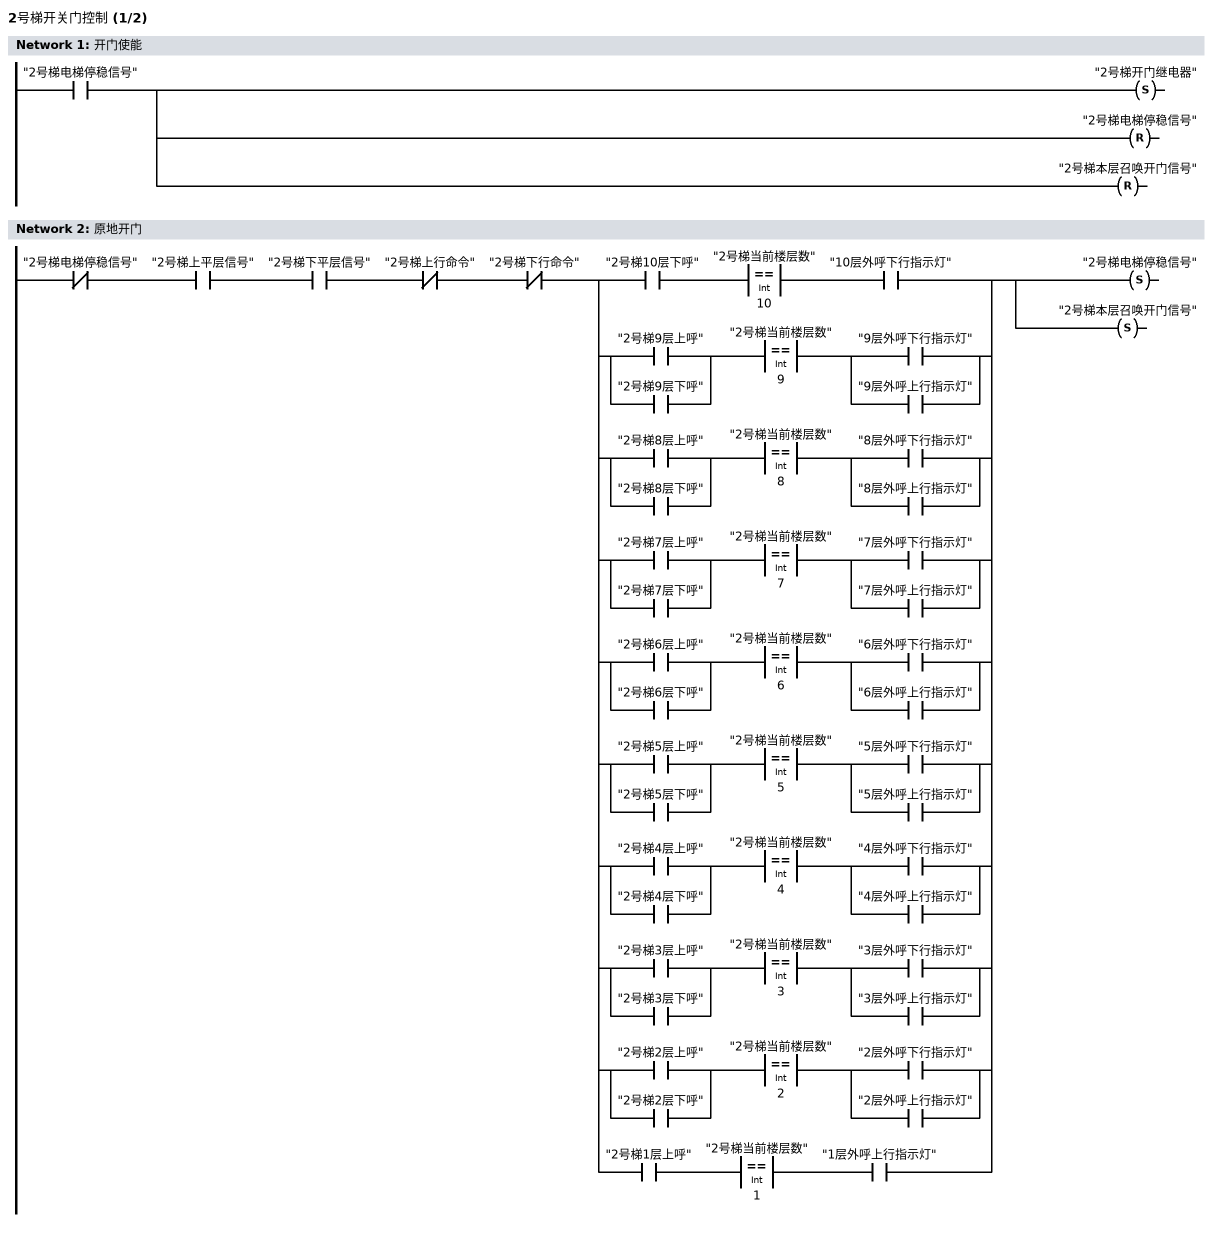
   RUNG wire#powerrail
      Contact( "2号梯电梯停稳信号" )
      wire#w1
      S_Coil( "2号梯开门继电器" )
   END_RUNG
   RUNG wire#w1
      R_Coil( "2号梯电梯停稳信号" )
   END_RUNG
   RUNG wire#w1
      R_Coil( "2号梯本层召唤开门信号" )
   END_RUNG
   // the same network as SCL:
   IF "2号梯电梯停稳信号" THEN "2号梯开门继电器" := TRUE; END_IF;
   #_w1 := "2号梯电梯停稳信号";
   IF #_w1 THEN
       "2号梯电梯停稳信号" := FALSE;
       "2号梯本层召唤开门信号" := FALSE;
   END_IF;
END_REGION

REGION Network 2: 原地开门
   RUNG wire#powerrail
      I_Contact( "2号梯电梯停稳信号" )
      Contact( "2号梯上平层信号" )
      Contact( "2号梯下平层信号" )
      I_Contact( "2号梯上行命令" )
      I_Contact( "2号梯下行命令" )
      wire#w1
      Contact( "2号梯10层下呼" )
      { S7_Templates := "SrcType := Int" } EQ_Contact(in1 := "2号梯当前楼层数", in2 := 10)
      Contact( "10层外呼下行指示灯" )
      wire#w2
      S_Coil( "2号梯电梯停稳信号" )
   END_RUNG
   RUNG wire#w1
      Contact( "2号梯9层上呼" )
      wire#w3
      { S7_Templates := "SrcType := Int" } EQ_Contact(in1 := "2号梯当前楼层数", in2 := 9)
      wire#w4
      Contact( "9层外呼下行指示灯" )
   END_RUNG wire#w2
   RUNG wire#w1
      Contact( "2号梯9层下呼" )
   END_RUNG wire#w3
   RUNG wire#w4
      Contact( "9层外呼上行指示灯" )
   END_RUNG wire#w2
   RUNG wire#w1
      Contact( "2号梯8层上呼" )
      wire#w5
      { S7_Templates := "SrcType := Int" } EQ_Contact(in1 := "2号梯当前楼层数", in2 := 8)
      wire#w6
      Contact( "8层外呼下行指示灯" )
   END_RUNG wire#w2
   RUNG wire#w1
      Contact( "2号梯8层下呼" )
   END_RUNG wire#w5
   RUNG wire#w6
      Contact( "8层外呼上行指示灯" )
   END_RUNG wire#w2
   RUNG wire#w1
      Contact( "2号梯7层上呼" )
      wire#w7
      { S7_Templates := "SrcType := Int" } EQ_Contact(in1 := "2号梯当前楼层数", in2 := 7)
      wire#w8
      Contact( "7层外呼下行指示灯" )
   END_RUNG wire#w2
   RUNG wire#w1
      Contact( "2号梯7层下呼" )
   END_RUNG wire#w7
   RUNG wire#w8
      Contact( "7层外呼上行指示灯" )
   END_RUNG wire#w2
   RUNG wire#w1
      Contact( "2号梯6层上呼" )
      wire#w9
      { S7_Templates := "SrcType := Int" } EQ_Contact(in1 := "2号梯当前楼层数", in2 := 6)
      wire#w10
      Contact( "6层外呼下行指示灯" )
   END_RUNG wire#w2
   RUNG wire#w1
      Contact( "2号梯6层下呼" )
   END_RUNG wire#w9
   RUNG wire#w10
      Contact( "6层外呼上行指示灯" )
   END_RUNG wire#w2
   RUNG wire#w1
      Contact( "2号梯5层上呼" )
      wire#w11
      { S7_Templates := "SrcType := Int" } EQ_Contact(in1 := "2号梯当前楼层数", in2 := 5)
      wire#w12
      Contact( "5层外呼下行指示灯" )
   END_RUNG wire#w2
   RUNG wire#w1
      Contact( "2号梯5层下呼" )
   END_RUNG wire#w11
   RUNG wire#w12
      Contact( "5层外呼上行指示灯" )
   END_RUNG wire#w2
   RUNG wire#w1
      Contact( "2号梯4层上呼" )
      wire#w13
      { S7_Templates := "SrcType := Int" } EQ_Contact(in1 := "2号梯当前楼层数", in2 := 4)
      wire#w14
      Contact( "4层外呼下行指示灯" )
   END_RUNG wire#w2
   RUNG wire#w1
      Contact( "2号梯4层下呼" )
   END_RUNG wire#w13
   RUNG wire#w14
      Contact( "4层外呼上行指示灯" )
   END_RUNG wire#w2
   RUNG wire#w1
      Contact( "2号梯3层上呼" )
      wire#w15
      { S7_Templates := "SrcType := Int" } EQ_Contact(in1 := "2号梯当前楼层数", in2 := 3)
      wire#w16
      Contact( "3层外呼下行指示灯" )
   END_RUNG wire#w2
   RUNG wire#w1
      Contact( "2号梯3层下呼" )
   END_RUNG wire#w15
   RUNG wire#w16
      Contact( "3层外呼上行指示灯" )
   END_RUNG wire#w2
   RUNG wire#w1
      Contact( "2号梯2层上呼" )
      wire#w17
      { S7_Templates := "SrcType := Int" } EQ_Contact(in1 := "2号梯当前楼层数", in2 := 2)
      wire#w18
      Contact( "2层外呼下行指示灯" )
   END_RUNG wire#w2
   RUNG wire#w1
      Contact( "2号梯2层下呼" )
   END_RUNG wire#w17
   RUNG wire#w18
      Contact( "2层外呼上行指示灯" )
   END_RUNG wire#w2
   RUNG wire#w1
      Contact( "2号梯1层上呼" )
      { S7_Templates := "SrcType := Int" } EQ_Contact(in1 := "2号梯当前楼层数", in2 := 1)
      Contact( "1层外呼上行指示灯" )
   END_RUNG wire#w2
   RUNG wire#w2
      S_Coil( "2号梯本层召唤开门信号" )
   END_RUNG
   // the same network as SCL:
   #_w1 := NOT "2号梯电梯停稳信号" AND "2号梯上平层信号" AND "2号梯下平层信号" AND NOT "2号梯上行命令" AND NOT "2号梯下行命令" AND (("2号梯10层下呼" AND ("2号梯当前楼层数" = 10) AND "10层外呼下行指示灯") OR (("2号梯9层上呼" OR "2号梯9层下呼") AND ("2号梯当前楼层数" = 9) AND ("9层外呼下行指示灯" OR "9层外呼上行指示灯")) OR (("2号梯8层上呼" OR "2号梯8层下呼") AND ("2号梯当前楼层数" = 8) AND ("8层外呼下行指示灯" OR "8层外呼上行指示灯")) OR (("2号梯7层上呼" OR "2号梯7层下呼") AND ("2号梯当前楼层数" = 7) AND ("7层外呼下行指示灯" OR "7层外呼上行指示灯")) OR (("2号梯6层上呼" OR "2号梯6层下呼") AND ("2号梯当前楼层数" = 6) AND ("6层外呼下行指示灯" OR "6层外呼上行指示灯")) OR (("2号梯5层上呼" OR "2号梯5层下呼") AND ("2号梯当前楼层数" = 5) AND ("5层外呼下行指示灯" OR "5层外呼上行指示灯")) OR (("2号梯4层上呼" OR "2号梯4层下呼") AND ("2号梯当前楼层数" = 4) AND ("4层外呼下行指示灯" OR "4层外呼上行指示灯")) OR (("2号梯3层上呼" OR "2号梯3层下呼") AND ("2号梯当前楼层数" = 3) AND ("3层外呼下行指示灯" OR "3层外呼上行指示灯")) OR (("2号梯2层上呼" OR "2号梯2层下呼") AND ("2号梯当前楼层数" = 2) AND ("2层外呼下行指示灯" OR "2层外呼上行指示灯")) OR ("2号梯1层上呼" AND ("2号梯当前楼层数" = 1) AND "1层外呼上行指示灯"));
   IF #_w1 THEN
       "2号梯电梯停稳信号" := TRUE;
       "2号梯本层召唤开门信号" := TRUE;
   END_IF;
END_REGION

REGION Network 3: 关门
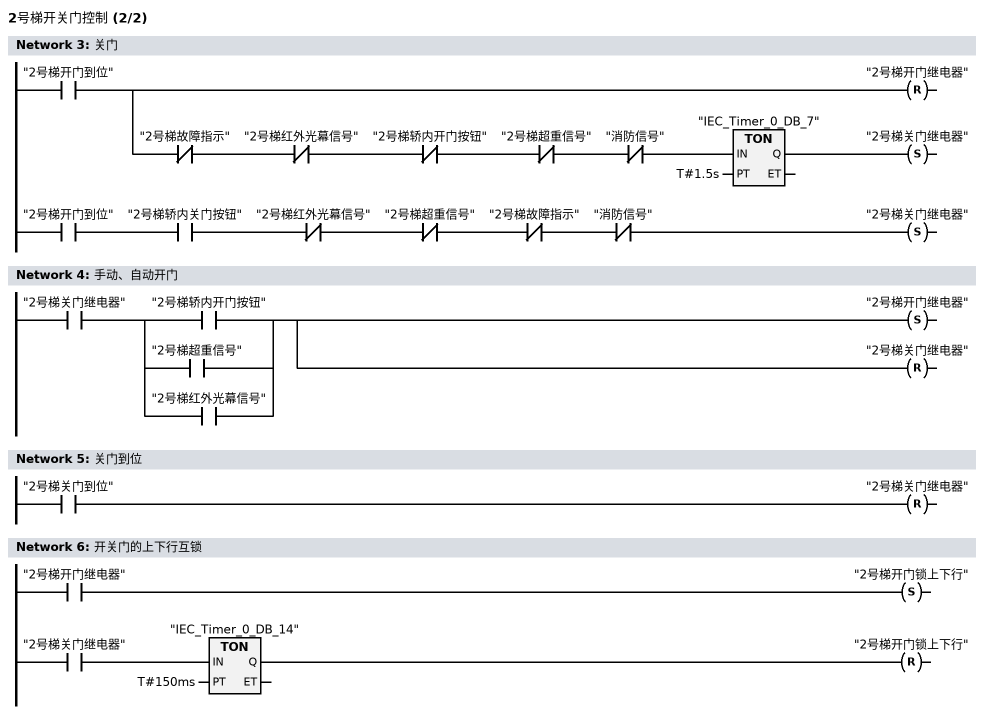
   IF "2号梯开门到位" THEN "2号梯开门继电器" := FALSE; END_IF;
   "IEC_Timer_0_DB_7".TON(IN := "2号梯开门到位" AND NOT "2号梯故障指示" AND NOT "2号梯红外光幕信号" AND NOT "2号梯轿内开门按钮" AND NOT "2号梯超重信号" AND NOT "消防信号",
                          PT := T#1.5s);
   IF "IEC_Timer_0_DB_7".Q THEN "2号梯关门继电器" := TRUE; END_IF;
   IF "2号梯开门到位" AND "2号梯轿内关门按钮" AND NOT "2号梯红外光幕信号" AND NOT "2号梯超重信号" AND NOT "2号梯故障指示" AND NOT "消防信号" THEN
       "2号梯关门继电器" := TRUE;
   END_IF;
END_REGION

REGION Network 4: 手动、自动开门
   RUNG wire#powerrail
      Contact( "2号梯关门继电器" )
      wire#w1
      Contact( "2号梯轿内开门按钮" )
      wire#w2
      S_Coil( "2号梯开门继电器" )
   END_RUNG
   RUNG wire#w1
      Contact( "2号梯超重信号" )
   END_RUNG wire#w2
   RUNG wire#w1
      Contact( "2号梯红外光幕信号" )
   END_RUNG wire#w2
   RUNG wire#w2
      R_Coil( "2号梯关门继电器" )
   END_RUNG
   // the same network as SCL:
   IF "2号梯关门继电器" AND ("2号梯轿内开门按钮" OR "2号梯超重信号" OR "2号梯红外光幕信号") THEN
       "2号梯开门继电器" := TRUE;
       "2号梯关门继电器" := FALSE;
   END_IF;
END_REGION

REGION Network 5: 关门到位
   RUNG wire#powerrail
      Contact( "2号梯关门到位" )
      R_Coil( "2号梯关门继电器" )
   END_RUNG
   // the same network as SCL:
   IF "2号梯关门到位" THEN "2号梯关门继电器" := FALSE; END_IF;
END_REGION

REGION Network 6: 开关门的上下行互锁
   IF "2号梯开门继电器" THEN "2号梯开门锁上下行" := TRUE; END_IF;
   "IEC_Timer_0_DB_14".TON(IN := "2号梯关门继电器", PT := T#150ms);
   IF "IEC_Timer_0_DB_14".Q THEN "2号梯开门锁上下行" := FALSE; END_IF;
END_REGION
END_FUNCTION

FUNCTION "1号梯开关门控制" : Void   // FC30, LAD
{ S7_Optimized_Access := 'TRUE' }
VERSION : 0.1
   VAR_TEMP   // added for the SCL form of the ladder/FBD networks
      _w1 : Bool;
   END_VAR
BEGIN

REGION Network 1: 开门使能
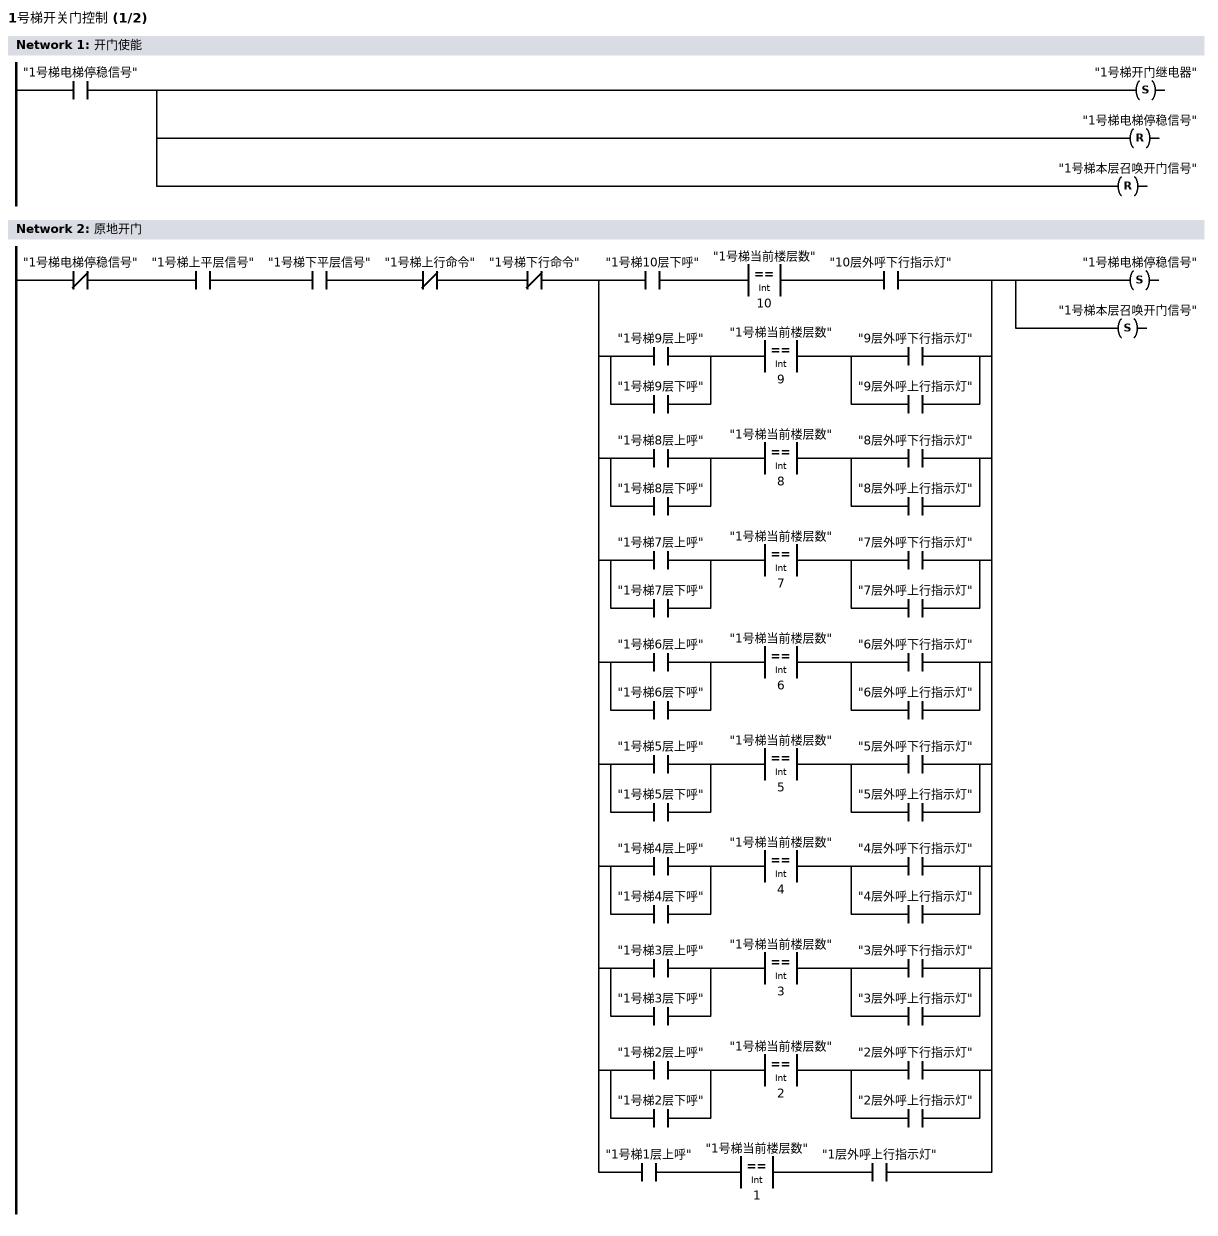
   RUNG wire#powerrail
      Contact( "1号梯电梯停稳信号" )
      wire#w1
      S_Coil( "1号梯开门继电器" )
   END_RUNG
   RUNG wire#w1
      R_Coil( "1号梯电梯停稳信号" )
   END_RUNG
   RUNG wire#w1
      R_Coil( "1号梯本层召唤开门信号" )
   END_RUNG
   // the same network as SCL:
   IF "1号梯电梯停稳信号" THEN "1号梯开门继电器" := TRUE; END_IF;
   #_w1 := "1号梯电梯停稳信号";
   IF #_w1 THEN
       "1号梯电梯停稳信号" := FALSE;
       "1号梯本层召唤开门信号" := FALSE;
   END_IF;
END_REGION

REGION Network 2: 原地开门
   RUNG wire#powerrail
      I_Contact( "1号梯电梯停稳信号" )
      Contact( "1号梯上平层信号" )
      Contact( "1号梯下平层信号" )
      I_Contact( "1号梯上行命令" )
      I_Contact( "1号梯下行命令" )
      wire#w1
      Contact( "1号梯10层下呼" )
      { S7_Templates := "SrcType := Int" } EQ_Contact(in1 := "1号梯当前楼层数", in2 := 10)
      Contact( "10层外呼下行指示灯" )
      wire#w2
      S_Coil( "1号梯电梯停稳信号" )
   END_RUNG
   RUNG wire#w1
      Contact( "1号梯9层上呼" )
      wire#w3
      { S7_Templates := "SrcType := Int" } EQ_Contact(in1 := "1号梯当前楼层数", in2 := 9)
      wire#w4
      Contact( "9层外呼下行指示灯" )
   END_RUNG wire#w2
   RUNG wire#w1
      Contact( "1号梯9层下呼" )
   END_RUNG wire#w3
   RUNG wire#w4
      Contact( "9层外呼上行指示灯" )
   END_RUNG wire#w2
   RUNG wire#w1
      Contact( "1号梯8层上呼" )
      wire#w5
      { S7_Templates := "SrcType := Int" } EQ_Contact(in1 := "1号梯当前楼层数", in2 := 8)
      wire#w6
      Contact( "8层外呼下行指示灯" )
   END_RUNG wire#w2
   RUNG wire#w1
      Contact( "1号梯8层下呼" )
   END_RUNG wire#w5
   RUNG wire#w6
      Contact( "8层外呼上行指示灯" )
   END_RUNG wire#w2
   RUNG wire#w1
      Contact( "1号梯7层上呼" )
      wire#w7
      { S7_Templates := "SrcType := Int" } EQ_Contact(in1 := "1号梯当前楼层数", in2 := 7)
      wire#w8
      Contact( "7层外呼下行指示灯" )
   END_RUNG wire#w2
   RUNG wire#w1
      Contact( "1号梯7层下呼" )
   END_RUNG wire#w7
   RUNG wire#w8
      Contact( "7层外呼上行指示灯" )
   END_RUNG wire#w2
   RUNG wire#w1
      Contact( "1号梯6层上呼" )
      wire#w9
      { S7_Templates := "SrcType := Int" } EQ_Contact(in1 := "1号梯当前楼层数", in2 := 6)
      wire#w10
      Contact( "6层外呼下行指示灯" )
   END_RUNG wire#w2
   RUNG wire#w1
      Contact( "1号梯6层下呼" )
   END_RUNG wire#w9
   RUNG wire#w10
      Contact( "6层外呼上行指示灯" )
   END_RUNG wire#w2
   RUNG wire#w1
      Contact( "1号梯5层上呼" )
      wire#w11
      { S7_Templates := "SrcType := Int" } EQ_Contact(in1 := "1号梯当前楼层数", in2 := 5)
      wire#w12
      Contact( "5层外呼下行指示灯" )
   END_RUNG wire#w2
   RUNG wire#w1
      Contact( "1号梯5层下呼" )
   END_RUNG wire#w11
   RUNG wire#w12
      Contact( "5层外呼上行指示灯" )
   END_RUNG wire#w2
   RUNG wire#w1
      Contact( "1号梯4层上呼" )
      wire#w13
      { S7_Templates := "SrcType := Int" } EQ_Contact(in1 := "1号梯当前楼层数", in2 := 4)
      wire#w14
      Contact( "4层外呼下行指示灯" )
   END_RUNG wire#w2
   RUNG wire#w1
      Contact( "1号梯4层下呼" )
   END_RUNG wire#w13
   RUNG wire#w14
      Contact( "4层外呼上行指示灯" )
   END_RUNG wire#w2
   RUNG wire#w1
      Contact( "1号梯3层上呼" )
      wire#w15
      { S7_Templates := "SrcType := Int" } EQ_Contact(in1 := "1号梯当前楼层数", in2 := 3)
      wire#w16
      Contact( "3层外呼下行指示灯" )
   END_RUNG wire#w2
   RUNG wire#w1
      Contact( "1号梯3层下呼" )
   END_RUNG wire#w15
   RUNG wire#w16
      Contact( "3层外呼上行指示灯" )
   END_RUNG wire#w2
   RUNG wire#w1
      Contact( "1号梯2层上呼" )
      wire#w17
      { S7_Templates := "SrcType := Int" } EQ_Contact(in1 := "1号梯当前楼层数", in2 := 2)
      wire#w18
      Contact( "2层外呼下行指示灯" )
   END_RUNG wire#w2
   RUNG wire#w1
      Contact( "1号梯2层下呼" )
   END_RUNG wire#w17
   RUNG wire#w18
      Contact( "2层外呼上行指示灯" )
   END_RUNG wire#w2
   RUNG wire#w1
      Contact( "1号梯1层上呼" )
      { S7_Templates := "SrcType := Int" } EQ_Contact(in1 := "1号梯当前楼层数", in2 := 1)
      Contact( "1层外呼上行指示灯" )
   END_RUNG wire#w2
   RUNG wire#w2
      S_Coil( "1号梯本层召唤开门信号" )
   END_RUNG
   // the same network as SCL:
   #_w1 := NOT "1号梯电梯停稳信号" AND "1号梯上平层信号" AND "1号梯下平层信号" AND NOT "1号梯上行命令" AND NOT "1号梯下行命令" AND (("1号梯10层下呼" AND ("1号梯当前楼层数" = 10) AND "10层外呼下行指示灯") OR (("1号梯9层上呼" OR "1号梯9层下呼") AND ("1号梯当前楼层数" = 9) AND ("9层外呼下行指示灯" OR "9层外呼上行指示灯")) OR (("1号梯8层上呼" OR "1号梯8层下呼") AND ("1号梯当前楼层数" = 8) AND ("8层外呼下行指示灯" OR "8层外呼上行指示灯")) OR (("1号梯7层上呼" OR "1号梯7层下呼") AND ("1号梯当前楼层数" = 7) AND ("7层外呼下行指示灯" OR "7层外呼上行指示灯")) OR (("1号梯6层上呼" OR "1号梯6层下呼") AND ("1号梯当前楼层数" = 6) AND ("6层外呼下行指示灯" OR "6层外呼上行指示灯")) OR (("1号梯5层上呼" OR "1号梯5层下呼") AND ("1号梯当前楼层数" = 5) AND ("5层外呼下行指示灯" OR "5层外呼上行指示灯")) OR (("1号梯4层上呼" OR "1号梯4层下呼") AND ("1号梯当前楼层数" = 4) AND ("4层外呼下行指示灯" OR "4层外呼上行指示灯")) OR (("1号梯3层上呼" OR "1号梯3层下呼") AND ("1号梯当前楼层数" = 3) AND ("3层外呼下行指示灯" OR "3层外呼上行指示灯")) OR (("1号梯2层上呼" OR "1号梯2层下呼") AND ("1号梯当前楼层数" = 2) AND ("2层外呼下行指示灯" OR "2层外呼上行指示灯")) OR ("1号梯1层上呼" AND ("1号梯当前楼层数" = 1) AND "1层外呼上行指示灯"));
   IF #_w1 THEN
       "1号梯电梯停稳信号" := TRUE;
       "1号梯本层召唤开门信号" := TRUE;
   END_IF;
END_REGION

REGION Network 3: 关门
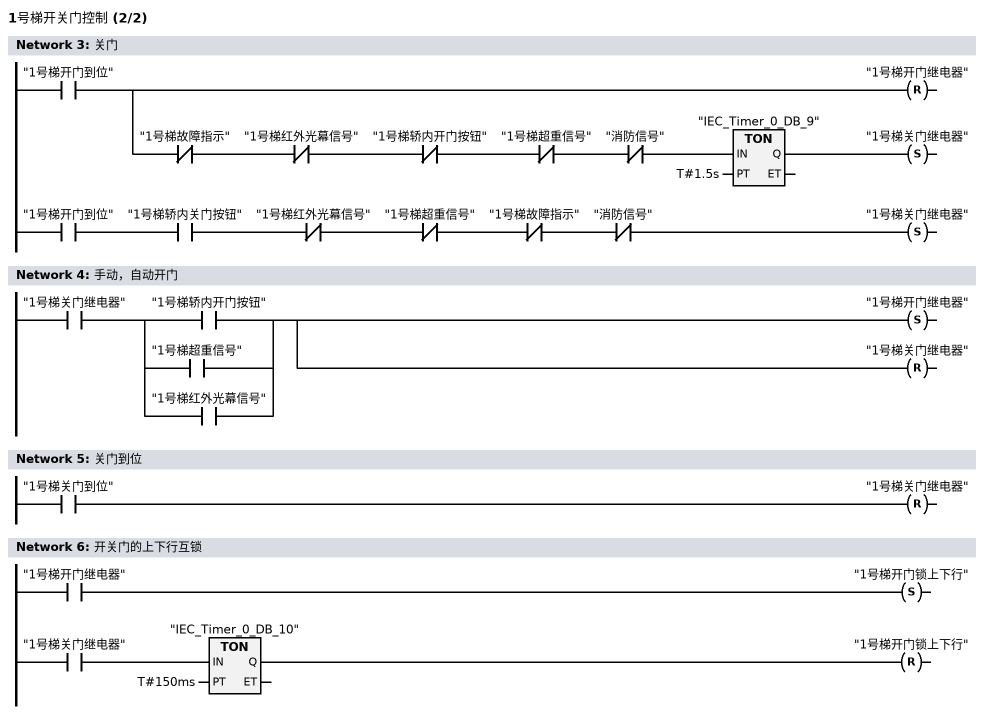
   IF "1号梯开门到位" THEN "1号梯开门继电器" := FALSE; END_IF;
   "IEC_Timer_0_DB_9".TON(IN := "1号梯开门到位" AND NOT "1号梯故障指示" AND NOT "1号梯红外光幕信号" AND NOT "1号梯轿内开门按钮" AND NOT "1号梯超重信号" AND NOT "消防信号",
                          PT := T#1.5s);
   IF "IEC_Timer_0_DB_9".Q THEN "1号梯关门继电器" := TRUE; END_IF;
   IF "1号梯开门到位" AND "1号梯轿内关门按钮" AND NOT "1号梯红外光幕信号" AND NOT "1号梯超重信号" AND NOT "1号梯故障指示" AND NOT "消防信号" THEN
       "1号梯关门继电器" := TRUE;
   END_IF;
END_REGION

REGION Network 4: 手动，自动开门
   RUNG wire#powerrail
      Contact( "1号梯关门继电器" )
      wire#w1
      Contact( "1号梯轿内开门按钮" )
      wire#w2
      S_Coil( "1号梯开门继电器" )
   END_RUNG
   RUNG wire#w1
      Contact( "1号梯超重信号" )
   END_RUNG wire#w2
   RUNG wire#w1
      Contact( "1号梯红外光幕信号" )
   END_RUNG wire#w2
   RUNG wire#w2
      R_Coil( "1号梯关门继电器" )
   END_RUNG
   // the same network as SCL:
   IF "1号梯关门继电器" AND ("1号梯轿内开门按钮" OR "1号梯超重信号" OR "1号梯红外光幕信号") THEN
       "1号梯开门继电器" := TRUE;
       "1号梯关门继电器" := FALSE;
   END_IF;
END_REGION

REGION Network 5: 关门到位
   RUNG wire#powerrail
      Contact( "1号梯关门到位" )
      R_Coil( "1号梯关门继电器" )
   END_RUNG
   // the same network as SCL:
   IF "1号梯关门到位" THEN "1号梯关门继电器" := FALSE; END_IF;
END_REGION

REGION Network 6: 开关门的上下行互锁
   IF "1号梯开门继电器" THEN "1号梯开门锁上下行" := TRUE; END_IF;
   "IEC_Timer_0_DB_10".TON(IN := "1号梯关门继电器", PT := T#150ms);
   IF "IEC_Timer_0_DB_10".Q THEN "1号梯开门锁上下行" := FALSE; END_IF;
END_REGION
END_FUNCTION

FUNCTION "3号梯目标楼层登记" : Void   // FC31, LAD
{ S7_Optimized_Access := 'TRUE' }
VERSION : 0.1
BEGIN

REGION Network 1: 楼层登记
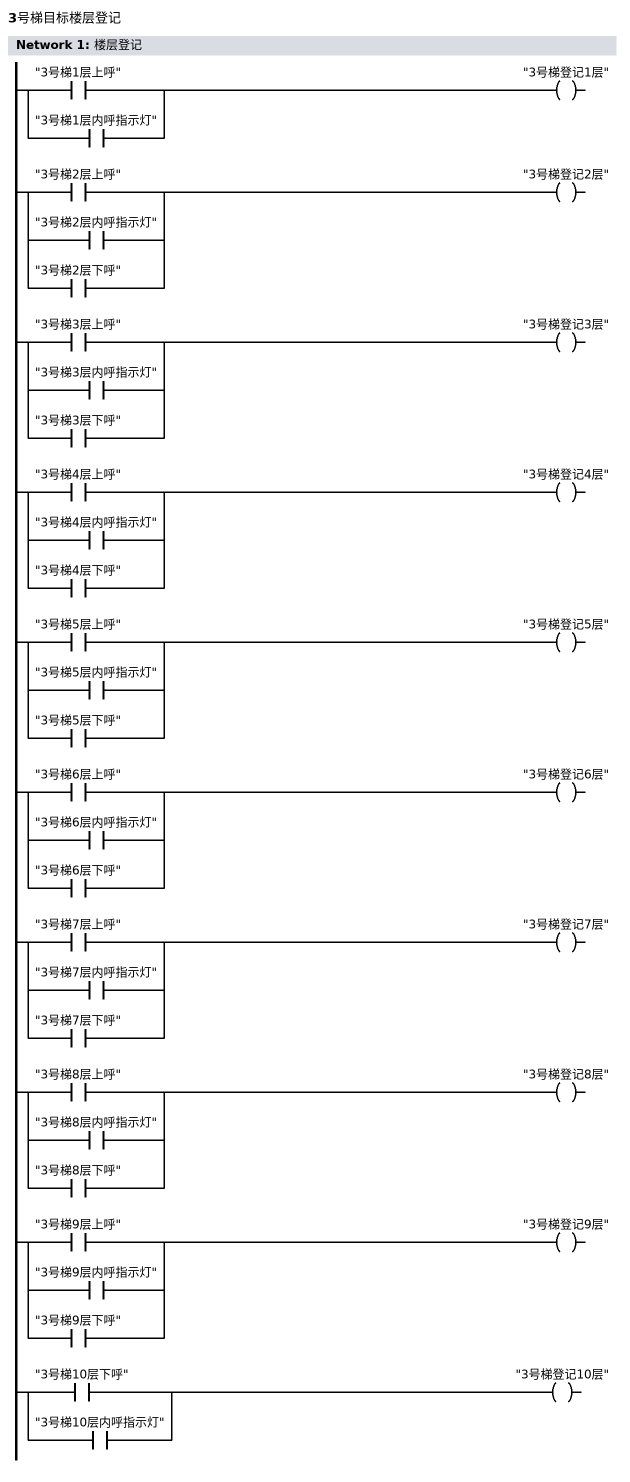
   RUNG wire#powerrail
      Contact( "3号梯1层上呼" )
      wire#w1
      Coil( "3号梯登记1层" )
   END_RUNG
   RUNG wire#powerrail
      Contact( "3号梯1层内呼指示灯" )
   END_RUNG wire#w1
   RUNG wire#powerrail
      Contact( "3号梯2层上呼" )
      wire#w2
      Coil( "3号梯登记2层" )
   END_RUNG
   RUNG wire#powerrail
      Contact( "3号梯2层内呼指示灯" )
   END_RUNG wire#w2
   RUNG wire#powerrail
      Contact( "3号梯2层下呼" )
   END_RUNG wire#w2
   RUNG wire#powerrail
      Contact( "3号梯3层上呼" )
      wire#w3
      Coil( "3号梯登记3层" )
   END_RUNG
   RUNG wire#powerrail
      Contact( "3号梯3层内呼指示灯" )
   END_RUNG wire#w3
   RUNG wire#powerrail
      Contact( "3号梯3层下呼" )
   END_RUNG wire#w3
   RUNG wire#powerrail
      Contact( "3号梯4层上呼" )
      wire#w4
      Coil( "3号梯登记4层" )
   END_RUNG
   RUNG wire#powerrail
      Contact( "3号梯4层内呼指示灯" )
   END_RUNG wire#w4
   RUNG wire#powerrail
      Contact( "3号梯4层下呼" )
   END_RUNG wire#w4
   RUNG wire#powerrail
      Contact( "3号梯5层上呼" )
      wire#w5
      Coil( "3号梯登记5层" )
   END_RUNG
   RUNG wire#powerrail
      Contact( "3号梯5层内呼指示灯" )
   END_RUNG wire#w5
   RUNG wire#powerrail
      Contact( "3号梯5层下呼" )
   END_RUNG wire#w5
   RUNG wire#powerrail
      Contact( "3号梯6层上呼" )
      wire#w6
      Coil( "3号梯登记6层" )
   END_RUNG
   RUNG wire#powerrail
      Contact( "3号梯6层内呼指示灯" )
   END_RUNG wire#w6
   RUNG wire#powerrail
      Contact( "3号梯6层下呼" )
   END_RUNG wire#w6
   RUNG wire#powerrail
      Contact( "3号梯7层上呼" )
      wire#w7
      Coil( "3号梯登记7层" )
   END_RUNG
   RUNG wire#powerrail
      Contact( "3号梯7层内呼指示灯" )
   END_RUNG wire#w7
   RUNG wire#powerrail
      Contact( "3号梯7层下呼" )
   END_RUNG wire#w7
   RUNG wire#powerrail
      Contact( "3号梯8层上呼" )
      wire#w8
      Coil( "3号梯登记8层" )
   END_RUNG
   RUNG wire#powerrail
      Contact( "3号梯8层内呼指示灯" )
   END_RUNG wire#w8
   RUNG wire#powerrail
      Contact( "3号梯8层下呼" )
   END_RUNG wire#w8
   RUNG wire#powerrail
      Contact( "3号梯9层上呼" )
      wire#w9
      Coil( "3号梯登记9层" )
   END_RUNG
   RUNG wire#powerrail
      Contact( "3号梯9层内呼指示灯" )
   END_RUNG wire#w9
   RUNG wire#powerrail
      Contact( "3号梯9层下呼" )
   END_RUNG wire#w9
   RUNG wire#powerrail
      Contact( "3号梯10层下呼" )
      wire#w10
      Coil( "3号梯登记10层" )
   END_RUNG
   RUNG wire#powerrail
      Contact( "3号梯10层内呼指示灯" )
   END_RUNG wire#w10
   // the same network as SCL:
   "3号梯登记1层" := "3号梯1层上呼" OR "3号梯1层内呼指示灯";
   "3号梯登记2层" := "3号梯2层上呼" OR "3号梯2层内呼指示灯" OR "3号梯2层下呼";
   "3号梯登记3层" := "3号梯3层上呼" OR "3号梯3层内呼指示灯" OR "3号梯3层下呼";
   "3号梯登记4层" := "3号梯4层上呼" OR "3号梯4层内呼指示灯" OR "3号梯4层下呼";
   "3号梯登记5层" := "3号梯5层上呼" OR "3号梯5层内呼指示灯" OR "3号梯5层下呼";
   "3号梯登记6层" := "3号梯6层上呼" OR "3号梯6层内呼指示灯" OR "3号梯6层下呼";
   "3号梯登记7层" := "3号梯7层上呼" OR "3号梯7层内呼指示灯" OR "3号梯7层下呼";
   "3号梯登记8层" := "3号梯8层上呼" OR "3号梯8层内呼指示灯" OR "3号梯8层下呼";
   "3号梯登记9层" := "3号梯9层上呼" OR "3号梯9层内呼指示灯" OR "3号梯9层下呼";
   "3号梯登记10层" := "3号梯10层下呼" OR "3号梯10层内呼指示灯";
END_REGION
END_FUNCTION

FUNCTION "2号梯目标楼层登记" : Void   // FC32, LAD
{ S7_Optimized_Access := 'TRUE' }
VERSION : 0.1
BEGIN

REGION Network 1: 楼层登记
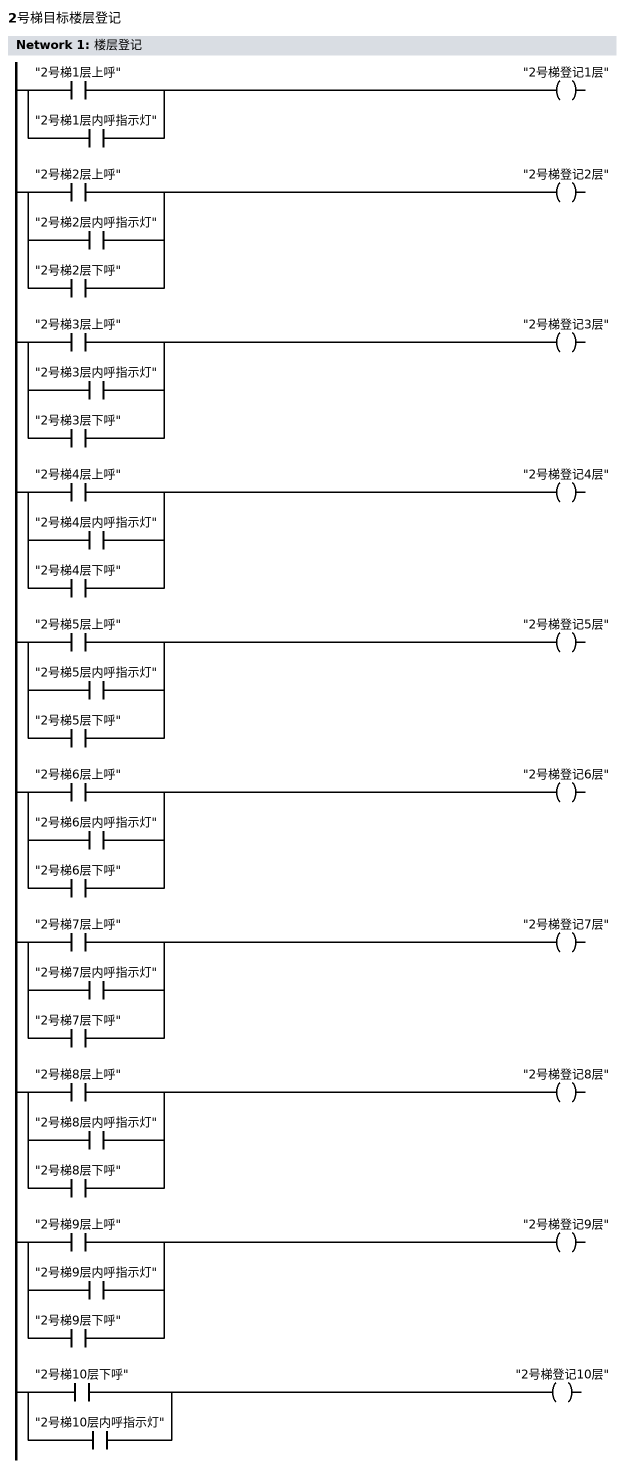
   RUNG wire#powerrail
      Contact( "2号梯1层上呼" )
      wire#w1
      Coil( "2号梯登记1层" )
   END_RUNG
   RUNG wire#powerrail
      Contact( "2号梯1层内呼指示灯" )
   END_RUNG wire#w1
   RUNG wire#powerrail
      Contact( "2号梯2层上呼" )
      wire#w2
      Coil( "2号梯登记2层" )
   END_RUNG
   RUNG wire#powerrail
      Contact( "2号梯2层内呼指示灯" )
   END_RUNG wire#w2
   RUNG wire#powerrail
      Contact( "2号梯2层下呼" )
   END_RUNG wire#w2
   RUNG wire#powerrail
      Contact( "2号梯3层上呼" )
      wire#w3
      Coil( "2号梯登记3层" )
   END_RUNG
   RUNG wire#powerrail
      Contact( "2号梯3层内呼指示灯" )
   END_RUNG wire#w3
   RUNG wire#powerrail
      Contact( "2号梯3层下呼" )
   END_RUNG wire#w3
   RUNG wire#powerrail
      Contact( "2号梯4层上呼" )
      wire#w4
      Coil( "2号梯登记4层" )
   END_RUNG
   RUNG wire#powerrail
      Contact( "2号梯4层内呼指示灯" )
   END_RUNG wire#w4
   RUNG wire#powerrail
      Contact( "2号梯4层下呼" )
   END_RUNG wire#w4
   RUNG wire#powerrail
      Contact( "2号梯5层上呼" )
      wire#w5
      Coil( "2号梯登记5层" )
   END_RUNG
   RUNG wire#powerrail
      Contact( "2号梯5层内呼指示灯" )
   END_RUNG wire#w5
   RUNG wire#powerrail
      Contact( "2号梯5层下呼" )
   END_RUNG wire#w5
   RUNG wire#powerrail
      Contact( "2号梯6层上呼" )
      wire#w6
      Coil( "2号梯登记6层" )
   END_RUNG
   RUNG wire#powerrail
      Contact( "2号梯6层内呼指示灯" )
   END_RUNG wire#w6
   RUNG wire#powerrail
      Contact( "2号梯6层下呼" )
   END_RUNG wire#w6
   RUNG wire#powerrail
      Contact( "2号梯7层上呼" )
      wire#w7
      Coil( "2号梯登记7层" )
   END_RUNG
   RUNG wire#powerrail
      Contact( "2号梯7层内呼指示灯" )
   END_RUNG wire#w7
   RUNG wire#powerrail
      Contact( "2号梯7层下呼" )
   END_RUNG wire#w7
   RUNG wire#powerrail
      Contact( "2号梯8层上呼" )
      wire#w8
      Coil( "2号梯登记8层" )
   END_RUNG
   RUNG wire#powerrail
      Contact( "2号梯8层内呼指示灯" )
   END_RUNG wire#w8
   RUNG wire#powerrail
      Contact( "2号梯8层下呼" )
   END_RUNG wire#w8
   RUNG wire#powerrail
      Contact( "2号梯9层上呼" )
      wire#w9
      Coil( "2号梯登记9层" )
   END_RUNG
   RUNG wire#powerrail
      Contact( "2号梯9层内呼指示灯" )
   END_RUNG wire#w9
   RUNG wire#powerrail
      Contact( "2号梯9层下呼" )
   END_RUNG wire#w9
   RUNG wire#powerrail
      Contact( "2号梯10层下呼" )
      wire#w10
      Coil( "2号梯登记10层" )
   END_RUNG
   RUNG wire#powerrail
      Contact( "2号梯10层内呼指示灯" )
   END_RUNG wire#w10
   // the same network as SCL:
   "2号梯登记1层" := "2号梯1层上呼" OR "2号梯1层内呼指示灯";
   "2号梯登记2层" := "2号梯2层上呼" OR "2号梯2层内呼指示灯" OR "2号梯2层下呼";
   "2号梯登记3层" := "2号梯3层上呼" OR "2号梯3层内呼指示灯" OR "2号梯3层下呼";
   "2号梯登记4层" := "2号梯4层上呼" OR "2号梯4层内呼指示灯" OR "2号梯4层下呼";
   "2号梯登记5层" := "2号梯5层上呼" OR "2号梯5层内呼指示灯" OR "2号梯5层下呼";
   "2号梯登记6层" := "2号梯6层上呼" OR "2号梯6层内呼指示灯" OR "2号梯6层下呼";
   "2号梯登记7层" := "2号梯7层上呼" OR "2号梯7层内呼指示灯" OR "2号梯7层下呼";
   "2号梯登记8层" := "2号梯8层上呼" OR "2号梯8层内呼指示灯" OR "2号梯8层下呼";
   "2号梯登记9层" := "2号梯9层上呼" OR "2号梯9层内呼指示灯" OR "2号梯9层下呼";
   "2号梯登记10层" := "2号梯10层下呼" OR "2号梯10层内呼指示灯";
END_REGION
END_FUNCTION

FUNCTION "3号梯自动选向" : Void   // FC33, LAD
{ S7_Optimized_Access := 'TRUE' }
VERSION : 0.1
BEGIN

REGION Network 1: 上行选向
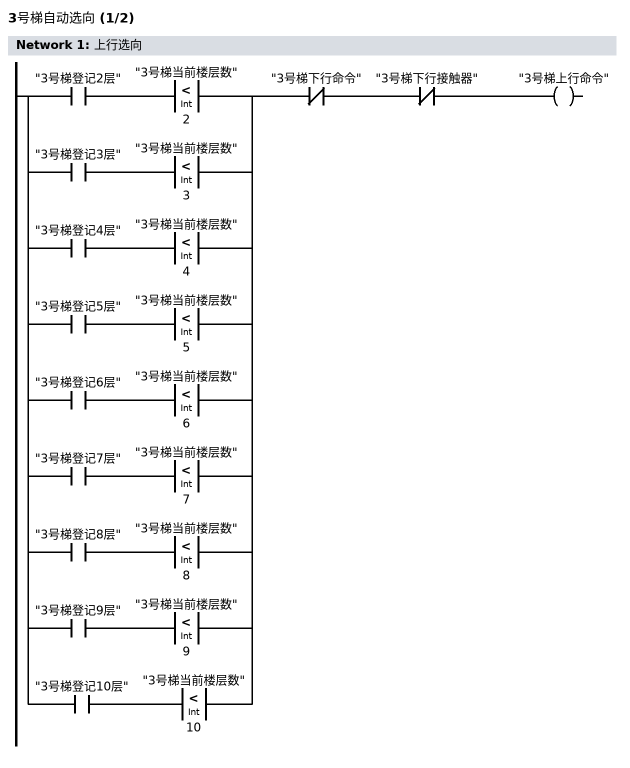
   RUNG wire#powerrail
      Contact( "3号梯登记2层" )
      { S7_Templates := "SrcType := Int" } LT_Contact(in1 := "3号梯当前楼层数", in2 := 2)
      wire#w1
      I_Contact( "3号梯下行命令" )
      I_Contact( "3号梯下行接触器" )
      Coil( "3号梯上行命令" )
   END_RUNG
   RUNG wire#powerrail
      Contact( "3号梯登记3层" )
      { S7_Templates := "SrcType := Int" } LT_Contact(in1 := "3号梯当前楼层数", in2 := 3)
   END_RUNG wire#w1
   RUNG wire#powerrail
      Contact( "3号梯登记4层" )
      { S7_Templates := "SrcType := Int" } LT_Contact(in1 := "3号梯当前楼层数", in2 := 4)
   END_RUNG wire#w1
   RUNG wire#powerrail
      Contact( "3号梯登记5层" )
      { S7_Templates := "SrcType := Int" } LT_Contact(in1 := "3号梯当前楼层数", in2 := 5)
   END_RUNG wire#w1
   RUNG wire#powerrail
      Contact( "3号梯登记6层" )
      { S7_Templates := "SrcType := Int" } LT_Contact(in1 := "3号梯当前楼层数", in2 := 6)
   END_RUNG wire#w1
   RUNG wire#powerrail
      Contact( "3号梯登记7层" )
      { S7_Templates := "SrcType := Int" } LT_Contact(in1 := "3号梯当前楼层数", in2 := 7)
   END_RUNG wire#w1
   RUNG wire#powerrail
      Contact( "3号梯登记8层" )
      { S7_Templates := "SrcType := Int" } LT_Contact(in1 := "3号梯当前楼层数", in2 := 8)
   END_RUNG wire#w1
   RUNG wire#powerrail
      Contact( "3号梯登记9层" )
      { S7_Templates := "SrcType := Int" } LT_Contact(in1 := "3号梯当前楼层数", in2 := 9)
   END_RUNG wire#w1
   RUNG wire#powerrail
      Contact( "3号梯登记10层" )
      { S7_Templates := "SrcType := Int" } LT_Contact(in1 := "3号梯当前楼层数", in2 := 10)
   END_RUNG wire#w1
   // the same network as SCL:
   "3号梯上行命令" := (("3号梯登记2层" AND ("3号梯当前楼层数" < 2)) OR ("3号梯登记3层" AND ("3号梯当前楼层数" < 3)) OR ("3号梯登记4层" AND ("3号梯当前楼层数" < 4)) OR ("3号梯登记5层" AND ("3号梯当前楼层数" < 5)) OR ("3号梯登记6层" AND ("3号梯当前楼层数" < 6)) OR ("3号梯登记7层" AND ("3号梯当前楼层数" < 7)) OR ("3号梯登记8层" AND ("3号梯当前楼层数" < 8)) OR ("3号梯登记9层" AND ("3号梯当前楼层数" < 9)) OR ("3号梯登记10层" AND ("3号梯当前楼层数" < 10))) AND NOT "3号梯下行命令" AND NOT "3号梯下行接触器";
END_REGION

REGION Network 2: 下行选向
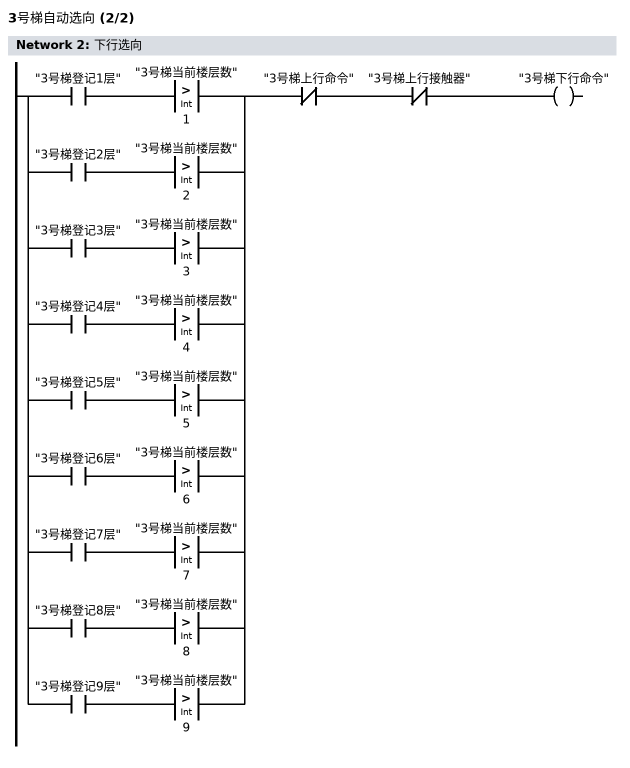
   RUNG wire#powerrail
      Contact( "3号梯登记1层" )
      { S7_Templates := "SrcType := Int" } GT_Contact(in1 := "3号梯当前楼层数", in2 := 1)
      wire#w1
      I_Contact( "3号梯上行命令" )
      I_Contact( "3号梯上行接触器" )
      Coil( "3号梯下行命令" )
   END_RUNG
   RUNG wire#powerrail
      Contact( "3号梯登记2层" )
      { S7_Templates := "SrcType := Int" } GT_Contact(in1 := "3号梯当前楼层数", in2 := 2)
   END_RUNG wire#w1
   RUNG wire#powerrail
      Contact( "3号梯登记3层" )
      { S7_Templates := "SrcType := Int" } GT_Contact(in1 := "3号梯当前楼层数", in2 := 3)
   END_RUNG wire#w1
   RUNG wire#powerrail
      Contact( "3号梯登记4层" )
      { S7_Templates := "SrcType := Int" } GT_Contact(in1 := "3号梯当前楼层数", in2 := 4)
   END_RUNG wire#w1
   RUNG wire#powerrail
      Contact( "3号梯登记5层" )
      { S7_Templates := "SrcType := Int" } GT_Contact(in1 := "3号梯当前楼层数", in2 := 5)
   END_RUNG wire#w1
   RUNG wire#powerrail
      Contact( "3号梯登记6层" )
      { S7_Templates := "SrcType := Int" } GT_Contact(in1 := "3号梯当前楼层数", in2 := 6)
   END_RUNG wire#w1
   RUNG wire#powerrail
      Contact( "3号梯登记7层" )
      { S7_Templates := "SrcType := Int" } GT_Contact(in1 := "3号梯当前楼层数", in2 := 7)
   END_RUNG wire#w1
   RUNG wire#powerrail
      Contact( "3号梯登记8层" )
      { S7_Templates := "SrcType := Int" } GT_Contact(in1 := "3号梯当前楼层数", in2 := 8)
   END_RUNG wire#w1
   RUNG wire#powerrail
      Contact( "3号梯登记9层" )
      { S7_Templates := "SrcType := Int" } GT_Contact(in1 := "3号梯当前楼层数", in2 := 9)
   END_RUNG wire#w1
   // the same network as SCL:
   "3号梯下行命令" := (("3号梯登记1层" AND ("3号梯当前楼层数" > 1)) OR ("3号梯登记2层" AND ("3号梯当前楼层数" > 2)) OR ("3号梯登记3层" AND ("3号梯当前楼层数" > 3)) OR ("3号梯登记4层" AND ("3号梯当前楼层数" > 4)) OR ("3号梯登记5层" AND ("3号梯当前楼层数" > 5)) OR ("3号梯登记6层" AND ("3号梯当前楼层数" > 6)) OR ("3号梯登记7层" AND ("3号梯当前楼层数" > 7)) OR ("3号梯登记8层" AND ("3号梯当前楼层数" > 8)) OR ("3号梯登记9层" AND ("3号梯当前楼层数" > 9))) AND NOT "3号梯上行命令" AND NOT "3号梯上行接触器";
END_REGION
END_FUNCTION

FUNCTION "2号梯自动选向" : Void   // FC34, LAD
{ S7_Optimized_Access := 'TRUE' }
VERSION : 0.1
BEGIN

REGION Network 1: 上行选向
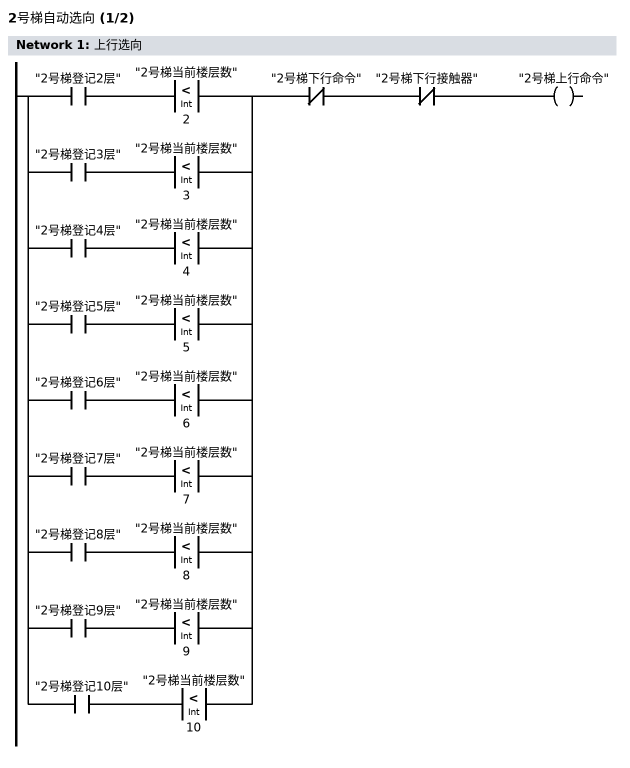
   RUNG wire#powerrail
      Contact( "2号梯登记2层" )
      { S7_Templates := "SrcType := Int" } LT_Contact(in1 := "2号梯当前楼层数", in2 := 2)
      wire#w1
      I_Contact( "2号梯下行命令" )
      I_Contact( "2号梯下行接触器" )
      Coil( "2号梯上行命令" )
   END_RUNG
   RUNG wire#powerrail
      Contact( "2号梯登记3层" )
      { S7_Templates := "SrcType := Int" } LT_Contact(in1 := "2号梯当前楼层数", in2 := 3)
   END_RUNG wire#w1
   RUNG wire#powerrail
      Contact( "2号梯登记4层" )
      { S7_Templates := "SrcType := Int" } LT_Contact(in1 := "2号梯当前楼层数", in2 := 4)
   END_RUNG wire#w1
   RUNG wire#powerrail
      Contact( "2号梯登记5层" )
      { S7_Templates := "SrcType := Int" } LT_Contact(in1 := "2号梯当前楼层数", in2 := 5)
   END_RUNG wire#w1
   RUNG wire#powerrail
      Contact( "2号梯登记6层" )
      { S7_Templates := "SrcType := Int" } LT_Contact(in1 := "2号梯当前楼层数", in2 := 6)
   END_RUNG wire#w1
   RUNG wire#powerrail
      Contact( "2号梯登记7层" )
      { S7_Templates := "SrcType := Int" } LT_Contact(in1 := "2号梯当前楼层数", in2 := 7)
   END_RUNG wire#w1
   RUNG wire#powerrail
      Contact( "2号梯登记8层" )
      { S7_Templates := "SrcType := Int" } LT_Contact(in1 := "2号梯当前楼层数", in2 := 8)
   END_RUNG wire#w1
   RUNG wire#powerrail
      Contact( "2号梯登记9层" )
      { S7_Templates := "SrcType := Int" } LT_Contact(in1 := "2号梯当前楼层数", in2 := 9)
   END_RUNG wire#w1
   RUNG wire#powerrail
      Contact( "2号梯登记10层" )
      { S7_Templates := "SrcType := Int" } LT_Contact(in1 := "2号梯当前楼层数", in2 := 10)
   END_RUNG wire#w1
   // the same network as SCL:
   "2号梯上行命令" := (("2号梯登记2层" AND ("2号梯当前楼层数" < 2)) OR ("2号梯登记3层" AND ("2号梯当前楼层数" < 3)) OR ("2号梯登记4层" AND ("2号梯当前楼层数" < 4)) OR ("2号梯登记5层" AND ("2号梯当前楼层数" < 5)) OR ("2号梯登记6层" AND ("2号梯当前楼层数" < 6)) OR ("2号梯登记7层" AND ("2号梯当前楼层数" < 7)) OR ("2号梯登记8层" AND ("2号梯当前楼层数" < 8)) OR ("2号梯登记9层" AND ("2号梯当前楼层数" < 9)) OR ("2号梯登记10层" AND ("2号梯当前楼层数" < 10))) AND NOT "2号梯下行命令" AND NOT "2号梯下行接触器";
END_REGION

REGION Network 2: 下行选向
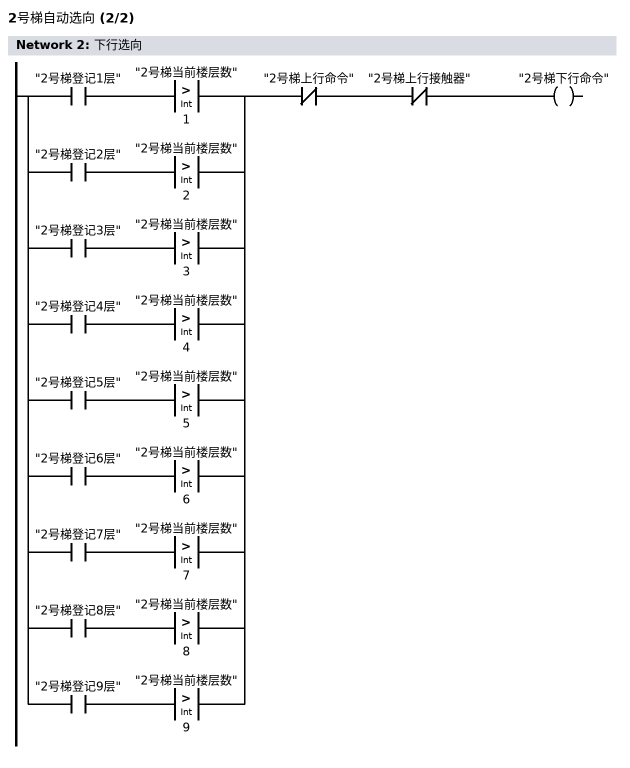
   RUNG wire#powerrail
      Contact( "2号梯登记1层" )
      { S7_Templates := "SrcType := Int" } GT_Contact(in1 := "2号梯当前楼层数", in2 := 1)
      wire#w1
      I_Contact( "2号梯上行命令" )
      I_Contact( "2号梯上行接触器" )
      Coil( "2号梯下行命令" )
   END_RUNG
   RUNG wire#powerrail
      Contact( "2号梯登记2层" )
      { S7_Templates := "SrcType := Int" } GT_Contact(in1 := "2号梯当前楼层数", in2 := 2)
   END_RUNG wire#w1
   RUNG wire#powerrail
      Contact( "2号梯登记3层" )
      { S7_Templates := "SrcType := Int" } GT_Contact(in1 := "2号梯当前楼层数", in2 := 3)
   END_RUNG wire#w1
   RUNG wire#powerrail
      Contact( "2号梯登记4层" )
      { S7_Templates := "SrcType := Int" } GT_Contact(in1 := "2号梯当前楼层数", in2 := 4)
   END_RUNG wire#w1
   RUNG wire#powerrail
      Contact( "2号梯登记5层" )
      { S7_Templates := "SrcType := Int" } GT_Contact(in1 := "2号梯当前楼层数", in2 := 5)
   END_RUNG wire#w1
   RUNG wire#powerrail
      Contact( "2号梯登记6层" )
      { S7_Templates := "SrcType := Int" } GT_Contact(in1 := "2号梯当前楼层数", in2 := 6)
   END_RUNG wire#w1
   RUNG wire#powerrail
      Contact( "2号梯登记7层" )
      { S7_Templates := "SrcType := Int" } GT_Contact(in1 := "2号梯当前楼层数", in2 := 7)
   END_RUNG wire#w1
   RUNG wire#powerrail
      Contact( "2号梯登记8层" )
      { S7_Templates := "SrcType := Int" } GT_Contact(in1 := "2号梯当前楼层数", in2 := 8)
   END_RUNG wire#w1
   RUNG wire#powerrail
      Contact( "2号梯登记9层" )
      { S7_Templates := "SrcType := Int" } GT_Contact(in1 := "2号梯当前楼层数", in2 := 9)
   END_RUNG wire#w1
   // the same network as SCL:
   "2号梯下行命令" := (("2号梯登记1层" AND ("2号梯当前楼层数" > 1)) OR ("2号梯登记2层" AND ("2号梯当前楼层数" > 2)) OR ("2号梯登记3层" AND ("2号梯当前楼层数" > 3)) OR ("2号梯登记4层" AND ("2号梯当前楼层数" > 4)) OR ("2号梯登记5层" AND ("2号梯当前楼层数" > 5)) OR ("2号梯登记6层" AND ("2号梯当前楼层数" > 6)) OR ("2号梯登记7层" AND ("2号梯当前楼层数" > 7)) OR ("2号梯登记8层" AND ("2号梯当前楼层数" > 8)) OR ("2号梯登记9层" AND ("2号梯当前楼层数" > 9))) AND NOT "2号梯上行命令" AND NOT "2号梯上行接触器";
END_REGION
END_FUNCTION

FUNCTION "3号梯启停" : Void   // FC35, LAD
{ S7_Optimized_Access := 'TRUE' }
VERSION : 0.1
   VAR_TEMP   // added for the SCL form of the ladder/FBD networks
      _w1 : Bool;
   END_VAR
BEGIN

REGION Network 1: 上行
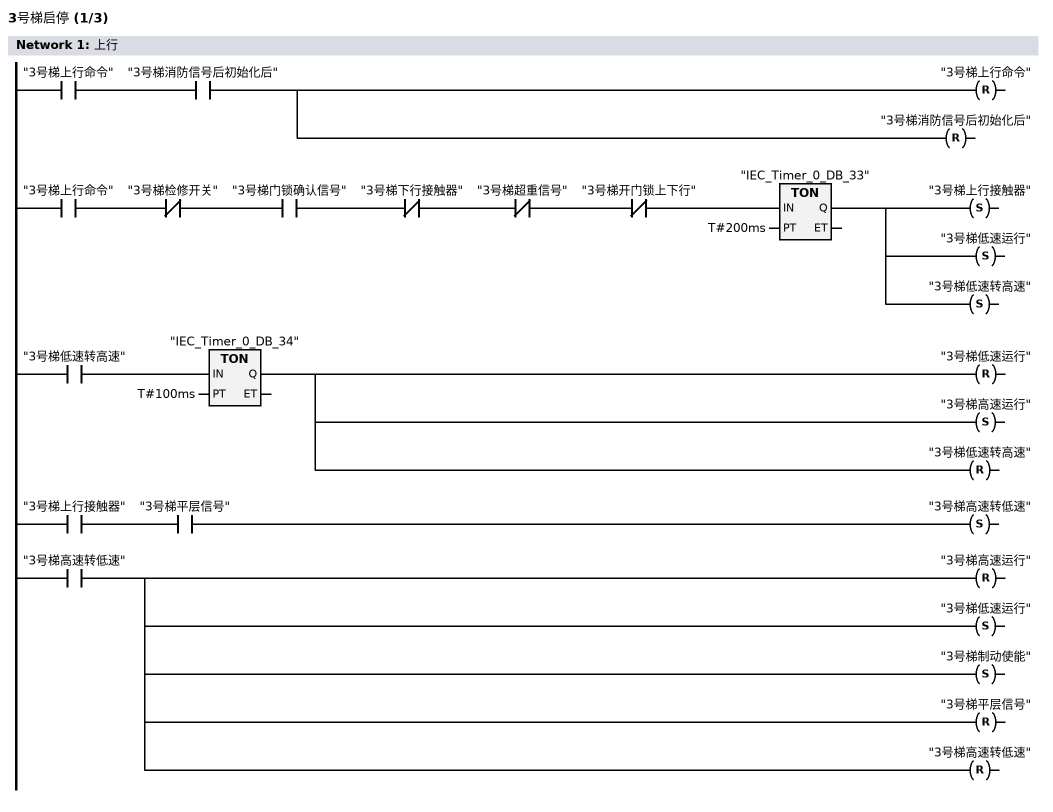
   #_w1 := "3号梯上行命令" AND "3号梯消防信号后初始化后";
   IF #_w1 THEN
       "3号梯上行命令" := FALSE;
       "3号梯消防信号后初始化后" := FALSE;
   END_IF;
   "IEC_Timer_0_DB_33".TON(IN := "3号梯上行命令" AND NOT "3号梯检修开关" AND "3号梯门锁确认信号" AND NOT "3号梯下行接触器" AND NOT "3号梯超重信号" AND NOT "3号梯开门锁上下行",
                           PT := T#200ms);
   IF "IEC_Timer_0_DB_33".Q THEN
       "3号梯上行接触器" := TRUE;
       "3号梯低速运行" := TRUE;
       "3号梯低速转高速" := TRUE;
   END_IF;
   "IEC_Timer_0_DB_34".TON(IN := "3号梯低速转高速", PT := T#100ms);
   IF "IEC_Timer_0_DB_34".Q THEN
       "3号梯低速运行" := FALSE;
       "3号梯高速运行" := TRUE;
       "3号梯低速转高速" := FALSE;
   END_IF;
   IF "3号梯上行接触器" AND "3号梯平层信号" THEN "3号梯高速转低速" := TRUE; END_IF;
   IF "3号梯高速转低速" THEN
       "3号梯高速运行" := FALSE;
       "3号梯低速运行" := TRUE;
       "3号梯制动使能" := TRUE;
       "3号梯平层信号" := FALSE;
       "3号梯高速转低速" := FALSE;
   END_IF;
END_REGION

REGION Network 2: 上行制动
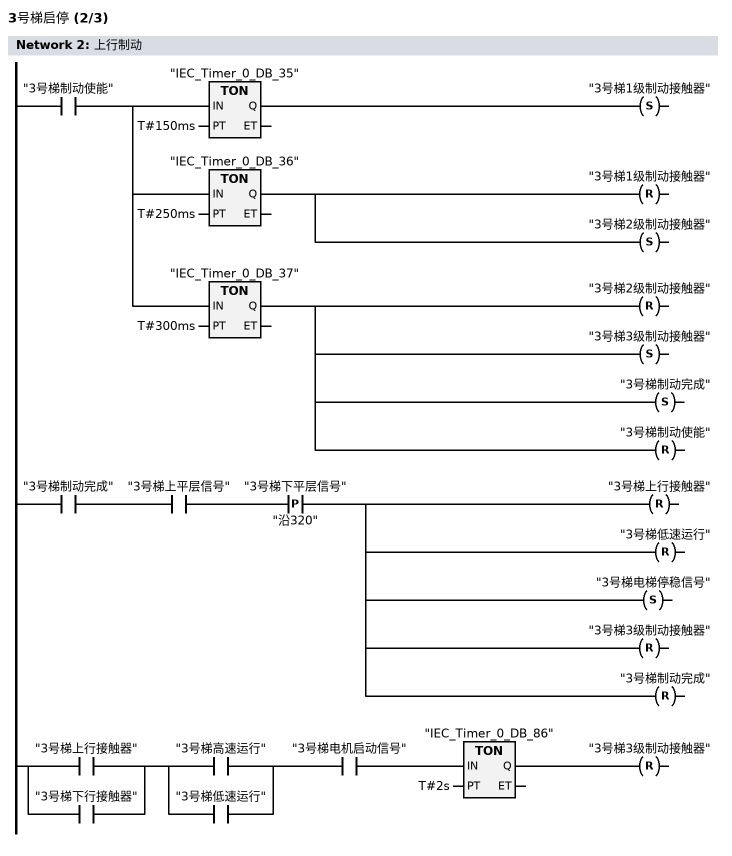
   "IEC_Timer_0_DB_35".TON(IN := "3号梯制动使能", PT := T#150ms);
   IF "IEC_Timer_0_DB_35".Q THEN "3号梯1级制动接触器" := TRUE; END_IF;
   "IEC_Timer_0_DB_36".TON(IN := "3号梯制动使能", PT := T#250ms);
   IF "IEC_Timer_0_DB_36".Q THEN
       "3号梯1级制动接触器" := FALSE;
       "3号梯2级制动接触器" := TRUE;
   END_IF;
   "IEC_Timer_0_DB_37".TON(IN := "3号梯制动使能", PT := T#300ms);
   IF "IEC_Timer_0_DB_37".Q THEN
       "3号梯2级制动接触器" := FALSE;
       "3号梯3级制动接触器" := TRUE;
       "3号梯制动完成" := TRUE;
       "3号梯制动使能" := FALSE;
   END_IF;
   #_w1 := "3号梯制动完成" AND "3号梯上平层信号" AND "3号梯下平层信号" AND NOT "沿320";   // rising edge of "3号梯下平层信号"
   "沿320" := "3号梯下平层信号";
   IF #_w1 THEN
       "3号梯上行接触器" := FALSE;
       "3号梯低速运行" := FALSE;
       "3号梯电梯停稳信号" := TRUE;
       "3号梯3级制动接触器" := FALSE;
       "3号梯制动完成" := FALSE;
   END_IF;
   "IEC_Timer_0_DB_86".TON(IN := ("3号梯上行接触器" OR "3号梯下行接触器") AND ("3号梯高速运行" OR "3号梯低速运行") AND "3号梯电机启动信号",
                           PT := T#2s);
   IF "IEC_Timer_0_DB_86".Q THEN "3号梯3级制动接触器" := FALSE; END_IF;
END_REGION

REGION Network 3: 下行
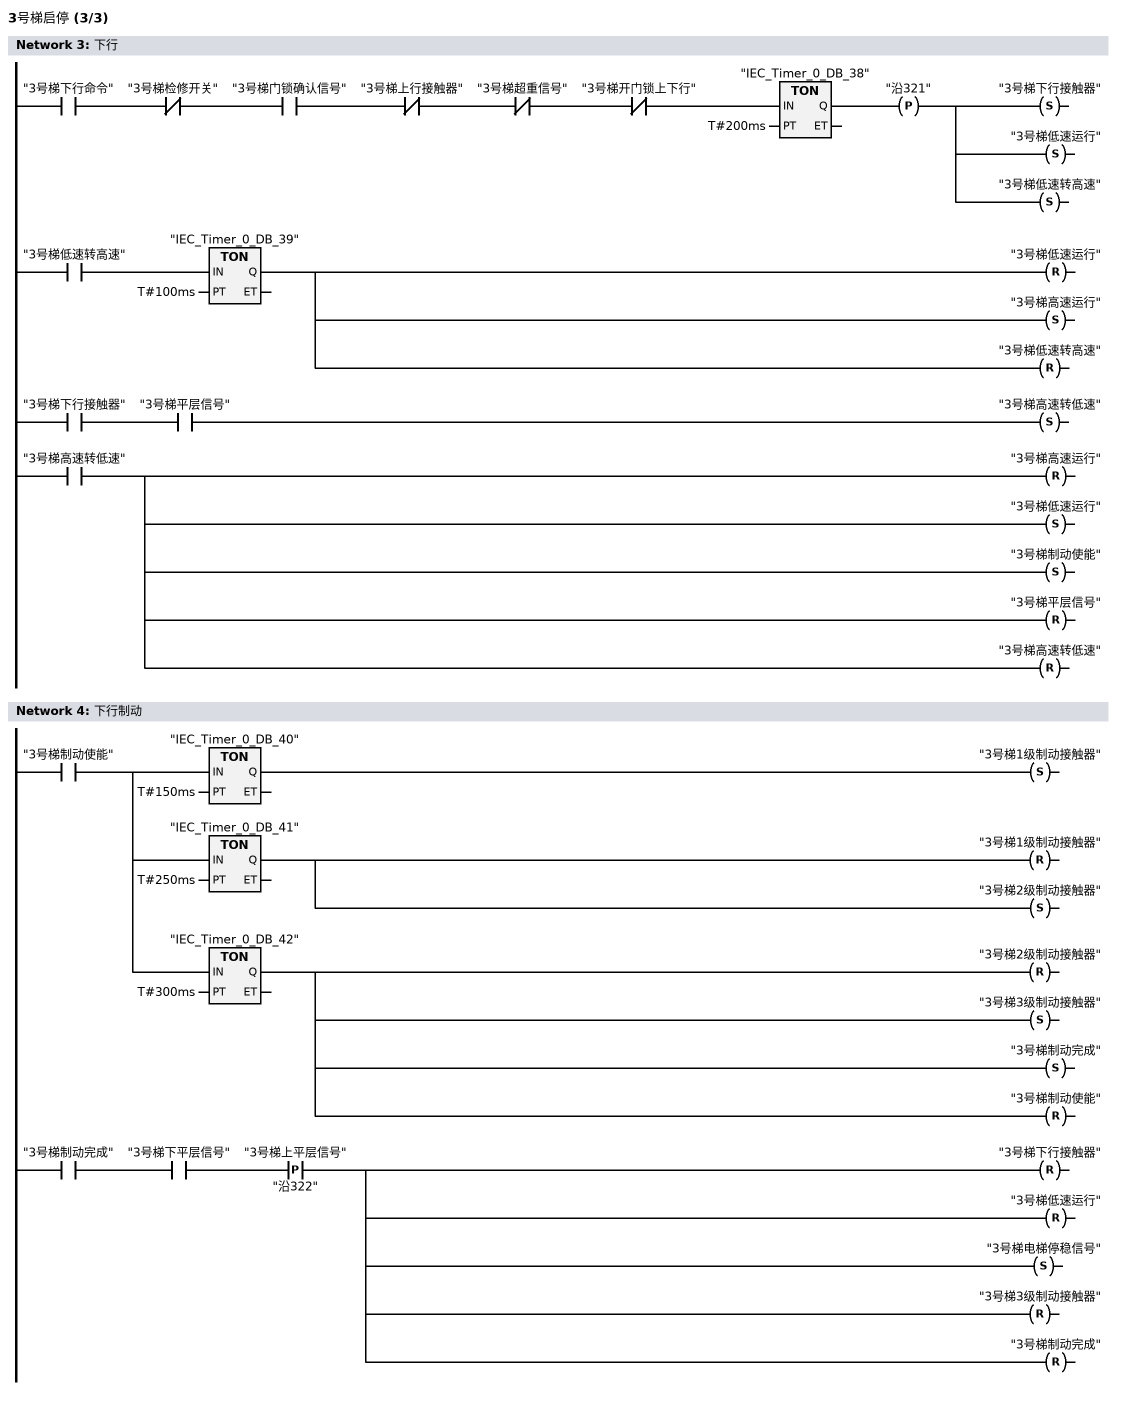
   "IEC_Timer_0_DB_38".TON(IN := "3号梯下行命令" AND NOT "3号梯检修开关" AND "3号梯门锁确认信号" AND NOT "3号梯上行接触器" AND NOT "3号梯超重信号" AND NOT "3号梯开门锁上下行",
                           PT := T#200ms);
   #_w1 := "IEC_Timer_0_DB_38".Q AND NOT "沿321";   // rising edge
   "沿321" := "IEC_Timer_0_DB_38".Q;
   IF #_w1 THEN
       "3号梯下行接触器" := TRUE;
       "3号梯低速运行" := TRUE;
       "3号梯低速转高速" := TRUE;
   END_IF;
   "IEC_Timer_0_DB_39".TON(IN := "3号梯低速转高速", PT := T#100ms);
   IF "IEC_Timer_0_DB_39".Q THEN
       "3号梯低速运行" := FALSE;
       "3号梯高速运行" := TRUE;
       "3号梯低速转高速" := FALSE;
   END_IF;
   IF "3号梯下行接触器" AND "3号梯平层信号" THEN "3号梯高速转低速" := TRUE; END_IF;
   IF "3号梯高速转低速" THEN
       "3号梯高速运行" := FALSE;
       "3号梯低速运行" := TRUE;
       "3号梯制动使能" := TRUE;
       "3号梯平层信号" := FALSE;
       "3号梯高速转低速" := FALSE;
   END_IF;
END_REGION

REGION Network 4: 下行制动
   "IEC_Timer_0_DB_40".TON(IN := "3号梯制动使能", PT := T#150ms);
   IF "IEC_Timer_0_DB_40".Q THEN "3号梯1级制动接触器" := TRUE; END_IF;
   "IEC_Timer_0_DB_41".TON(IN := "3号梯制动使能", PT := T#250ms);
   IF "IEC_Timer_0_DB_41".Q THEN
       "3号梯1级制动接触器" := FALSE;
       "3号梯2级制动接触器" := TRUE;
   END_IF;
   "IEC_Timer_0_DB_42".TON(IN := "3号梯制动使能", PT := T#300ms);
   IF "IEC_Timer_0_DB_42".Q THEN
       "3号梯2级制动接触器" := FALSE;
       "3号梯3级制动接触器" := TRUE;
       "3号梯制动完成" := TRUE;
       "3号梯制动使能" := FALSE;
   END_IF;
   #_w1 := "3号梯制动完成" AND "3号梯下平层信号" AND "3号梯上平层信号" AND NOT "沿322";   // rising edge of "3号梯上平层信号"
   "沿322" := "3号梯上平层信号";
   IF #_w1 THEN
       "3号梯下行接触器" := FALSE;
       "3号梯低速运行" := FALSE;
       "3号梯电梯停稳信号" := TRUE;
       "3号梯3级制动接触器" := FALSE;
       "3号梯制动完成" := FALSE;
   END_IF;
END_REGION
END_FUNCTION

FUNCTION "2号梯启停" : Void   // FC36, LAD
{ S7_Optimized_Access := 'TRUE' }
VERSION : 0.1
   VAR_TEMP   // added for the SCL form of the ladder/FBD networks
      _w1 : Bool;
   END_VAR
BEGIN

REGION Network 1: 上行
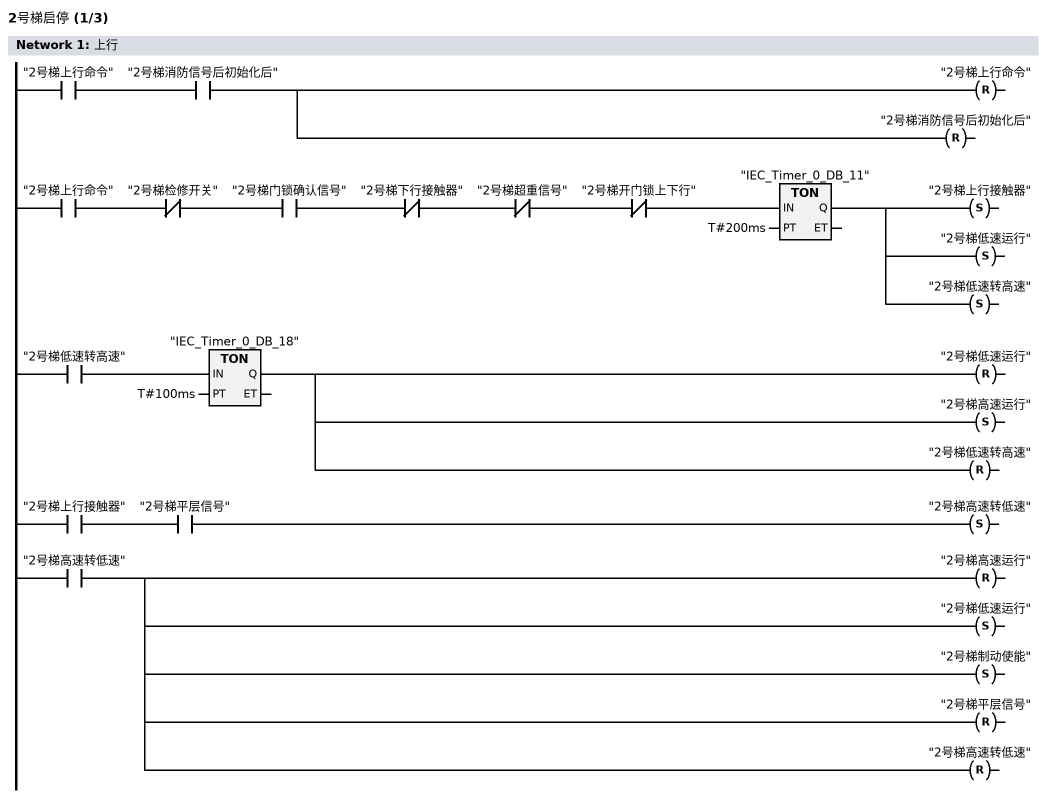
   #_w1 := "2号梯上行命令" AND "2号梯消防信号后初始化后";
   IF #_w1 THEN
       "2号梯上行命令" := FALSE;
       "2号梯消防信号后初始化后" := FALSE;
   END_IF;
   "IEC_Timer_0_DB_11".TON(IN := "2号梯上行命令" AND NOT "2号梯检修开关" AND "2号梯门锁确认信号" AND NOT "2号梯下行接触器" AND NOT "2号梯超重信号" AND NOT "2号梯开门锁上下行",
                           PT := T#200ms);
   IF "IEC_Timer_0_DB_11".Q THEN
       "2号梯上行接触器" := TRUE;
       "2号梯低速运行" := TRUE;
       "2号梯低速转高速" := TRUE;
   END_IF;
   "IEC_Timer_0_DB_18".TON(IN := "2号梯低速转高速", PT := T#100ms);
   IF "IEC_Timer_0_DB_18".Q THEN
       "2号梯低速运行" := FALSE;
       "2号梯高速运行" := TRUE;
       "2号梯低速转高速" := FALSE;
   END_IF;
   IF "2号梯上行接触器" AND "2号梯平层信号" THEN "2号梯高速转低速" := TRUE; END_IF;
   IF "2号梯高速转低速" THEN
       "2号梯高速运行" := FALSE;
       "2号梯低速运行" := TRUE;
       "2号梯制动使能" := TRUE;
       "2号梯平层信号" := FALSE;
       "2号梯高速转低速" := FALSE;
   END_IF;
END_REGION

REGION Network 2: 上行制动
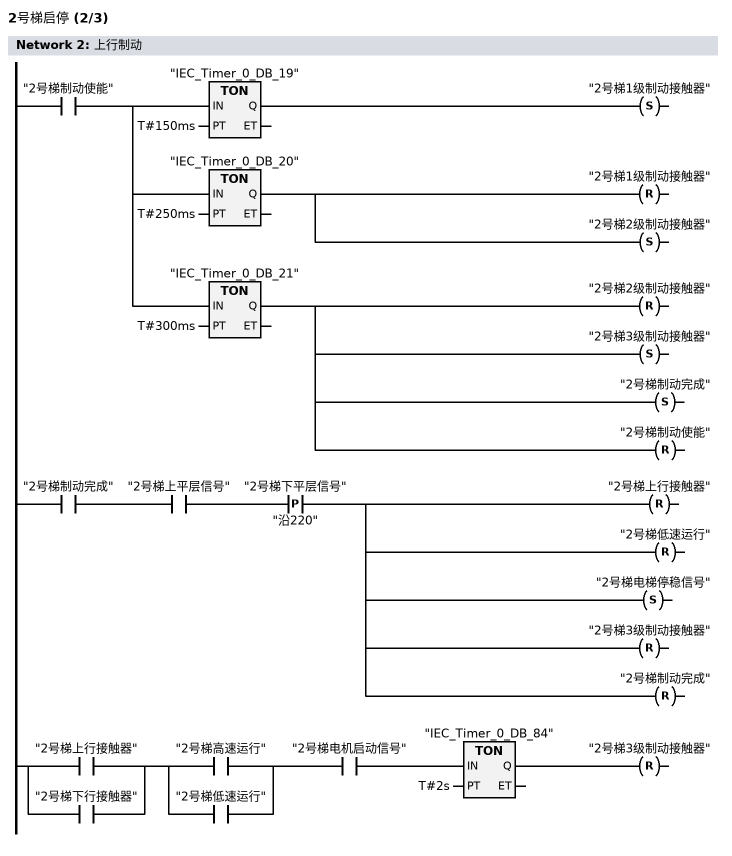
   "IEC_Timer_0_DB_19".TON(IN := "2号梯制动使能", PT := T#150ms);
   IF "IEC_Timer_0_DB_19".Q THEN "2号梯1级制动接触器" := TRUE; END_IF;
   "IEC_Timer_0_DB_20".TON(IN := "2号梯制动使能", PT := T#250ms);
   IF "IEC_Timer_0_DB_20".Q THEN
       "2号梯1级制动接触器" := FALSE;
       "2号梯2级制动接触器" := TRUE;
   END_IF;
   "IEC_Timer_0_DB_21".TON(IN := "2号梯制动使能", PT := T#300ms);
   IF "IEC_Timer_0_DB_21".Q THEN
       "2号梯2级制动接触器" := FALSE;
       "2号梯3级制动接触器" := TRUE;
       "2号梯制动完成" := TRUE;
       "2号梯制动使能" := FALSE;
   END_IF;
   #_w1 := "2号梯制动完成" AND "2号梯上平层信号" AND "2号梯下平层信号" AND NOT "沿220";   // rising edge of "2号梯下平层信号"
   "沿220" := "2号梯下平层信号";
   IF #_w1 THEN
       "2号梯上行接触器" := FALSE;
       "2号梯低速运行" := FALSE;
       "2号梯电梯停稳信号" := TRUE;
       "2号梯3级制动接触器" := FALSE;
       "2号梯制动完成" := FALSE;
   END_IF;
   "IEC_Timer_0_DB_84".TON(IN := ("2号梯上行接触器" OR "2号梯下行接触器") AND ("2号梯高速运行" OR "2号梯低速运行") AND "2号梯电机启动信号",
                           PT := T#2s);
   IF "IEC_Timer_0_DB_84".Q THEN "2号梯3级制动接触器" := FALSE; END_IF;
END_REGION

REGION Network 3: 下行
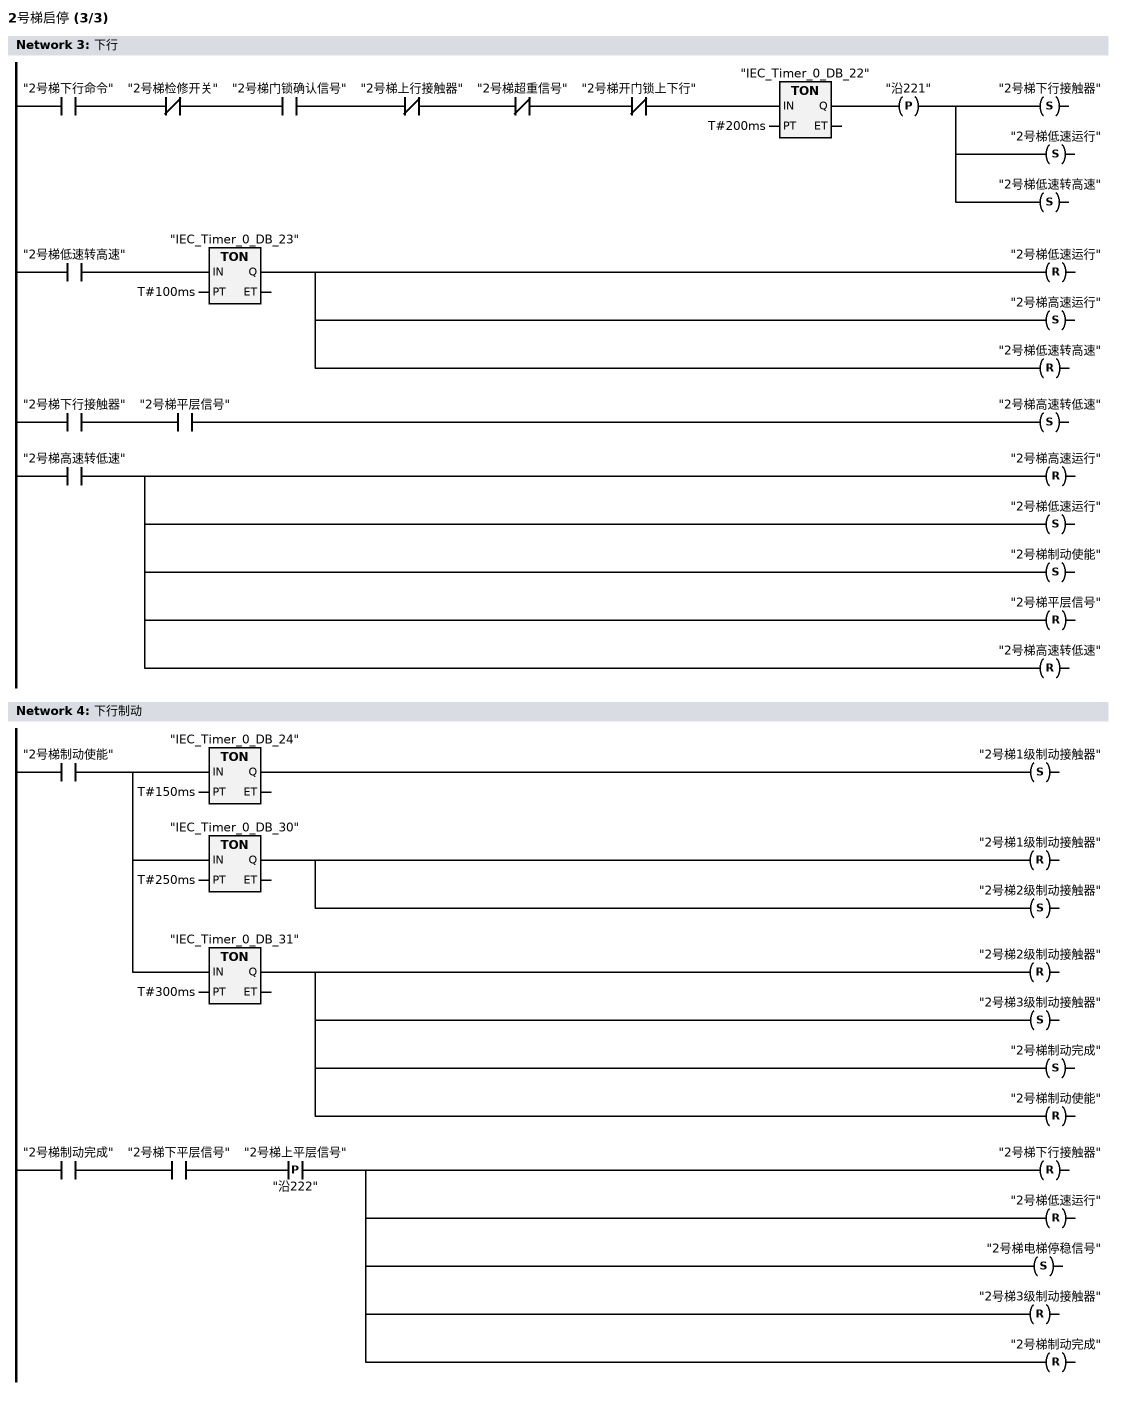
   "IEC_Timer_0_DB_22".TON(IN := "2号梯下行命令" AND NOT "2号梯检修开关" AND "2号梯门锁确认信号" AND NOT "2号梯上行接触器" AND NOT "2号梯超重信号" AND NOT "2号梯开门锁上下行",
                           PT := T#200ms);
   #_w1 := "IEC_Timer_0_DB_22".Q AND NOT "沿221";   // rising edge
   "沿221" := "IEC_Timer_0_DB_22".Q;
   IF #_w1 THEN
       "2号梯下行接触器" := TRUE;
       "2号梯低速运行" := TRUE;
       "2号梯低速转高速" := TRUE;
   END_IF;
   "IEC_Timer_0_DB_23".TON(IN := "2号梯低速转高速", PT := T#100ms);
   IF "IEC_Timer_0_DB_23".Q THEN
       "2号梯低速运行" := FALSE;
       "2号梯高速运行" := TRUE;
       "2号梯低速转高速" := FALSE;
   END_IF;
   IF "2号梯下行接触器" AND "2号梯平层信号" THEN "2号梯高速转低速" := TRUE; END_IF;
   IF "2号梯高速转低速" THEN
       "2号梯高速运行" := FALSE;
       "2号梯低速运行" := TRUE;
       "2号梯制动使能" := TRUE;
       "2号梯平层信号" := FALSE;
       "2号梯高速转低速" := FALSE;
   END_IF;
END_REGION

REGION Network 4: 下行制动
   "IEC_Timer_0_DB_24".TON(IN := "2号梯制动使能", PT := T#150ms);
   IF "IEC_Timer_0_DB_24".Q THEN "2号梯1级制动接触器" := TRUE; END_IF;
   "IEC_Timer_0_DB_30".TON(IN := "2号梯制动使能", PT := T#250ms);
   IF "IEC_Timer_0_DB_30".Q THEN
       "2号梯1级制动接触器" := FALSE;
       "2号梯2级制动接触器" := TRUE;
   END_IF;
   "IEC_Timer_0_DB_31".TON(IN := "2号梯制动使能", PT := T#300ms);
   IF "IEC_Timer_0_DB_31".Q THEN
       "2号梯2级制动接触器" := FALSE;
       "2号梯3级制动接触器" := TRUE;
       "2号梯制动完成" := TRUE;
       "2号梯制动使能" := FALSE;
   END_IF;
   #_w1 := "2号梯制动完成" AND "2号梯下平层信号" AND "2号梯上平层信号" AND NOT "沿222";   // rising edge of "2号梯上平层信号"
   "沿222" := "2号梯上平层信号";
   IF #_w1 THEN
       "2号梯下行接触器" := FALSE;
       "2号梯低速运行" := FALSE;
       "2号梯电梯停稳信号" := TRUE;
       "2号梯3级制动接触器" := FALSE;
       "2号梯制动完成" := FALSE;
   END_IF;
END_REGION
END_FUNCTION

FUNCTION "2号梯顺向截梯" : Void   // FC37, LAD
{ S7_Optimized_Access := 'TRUE' }
VERSION : 0.1
BEGIN

REGION Network 1: 上行拦截电梯
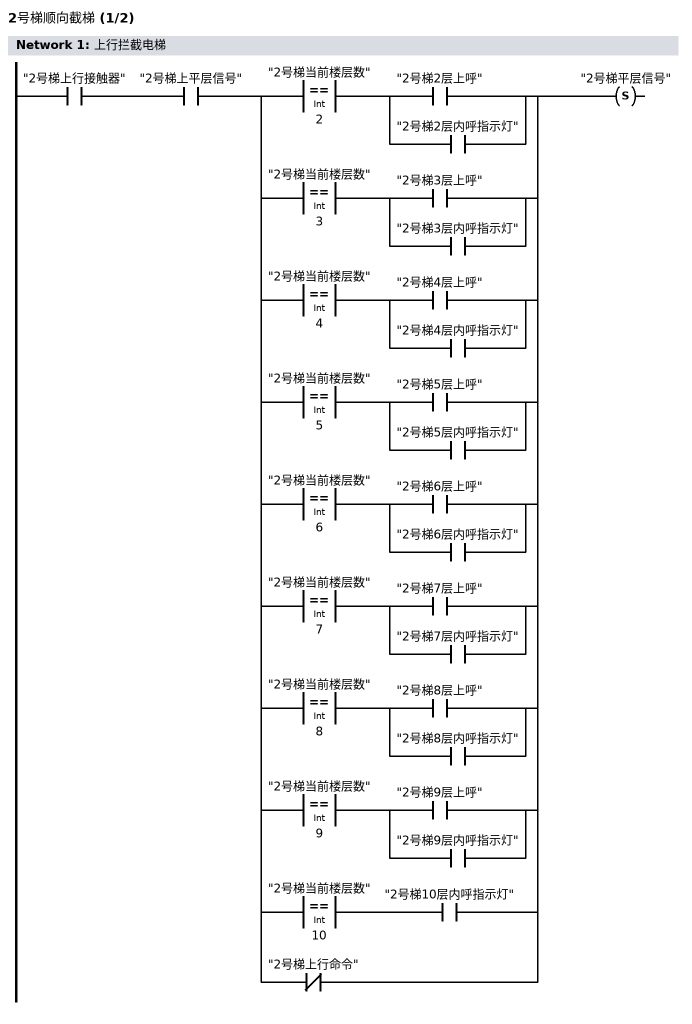
   RUNG wire#powerrail
      Contact( "2号梯上行接触器" )
      Contact( "2号梯上平层信号" )
      wire#w1
      { S7_Templates := "SrcType := Int" } EQ_Contact(in1 := "2号梯当前楼层数", in2 := 2)
      wire#w2
      Contact( "2号梯2层上呼" )
      wire#w3
      S_Coil( "2号梯平层信号" )
   END_RUNG
   RUNG wire#w2
      Contact( "2号梯2层内呼指示灯" )
   END_RUNG wire#w3
   RUNG wire#w1
      { S7_Templates := "SrcType := Int" } EQ_Contact(in1 := "2号梯当前楼层数", in2 := 3)
      wire#w4
      Contact( "2号梯3层上呼" )
   END_RUNG wire#w3
   RUNG wire#w4
      Contact( "2号梯3层内呼指示灯" )
   END_RUNG wire#w3
   RUNG wire#w1
      { S7_Templates := "SrcType := Int" } EQ_Contact(in1 := "2号梯当前楼层数", in2 := 4)
      wire#w5
      Contact( "2号梯4层上呼" )
   END_RUNG wire#w3
   RUNG wire#w5
      Contact( "2号梯4层内呼指示灯" )
   END_RUNG wire#w3
   RUNG wire#w1
      { S7_Templates := "SrcType := Int" } EQ_Contact(in1 := "2号梯当前楼层数", in2 := 5)
      wire#w6
      Contact( "2号梯5层上呼" )
   END_RUNG wire#w3
   RUNG wire#w6
      Contact( "2号梯5层内呼指示灯" )
   END_RUNG wire#w3
   RUNG wire#w1
      { S7_Templates := "SrcType := Int" } EQ_Contact(in1 := "2号梯当前楼层数", in2 := 6)
      wire#w7
      Contact( "2号梯6层上呼" )
   END_RUNG wire#w3
   RUNG wire#w7
      Contact( "2号梯6层内呼指示灯" )
   END_RUNG wire#w3
   RUNG wire#w1
      { S7_Templates := "SrcType := Int" } EQ_Contact(in1 := "2号梯当前楼层数", in2 := 7)
      wire#w8
      Contact( "2号梯7层上呼" )
   END_RUNG wire#w3
   RUNG wire#w8
      Contact( "2号梯7层内呼指示灯" )
   END_RUNG wire#w3
   RUNG wire#w1
      { S7_Templates := "SrcType := Int" } EQ_Contact(in1 := "2号梯当前楼层数", in2 := 8)
      wire#w9
      Contact( "2号梯8层上呼" )
   END_RUNG wire#w3
   RUNG wire#w9
      Contact( "2号梯8层内呼指示灯" )
   END_RUNG wire#w3
   RUNG wire#w1
      { S7_Templates := "SrcType := Int" } EQ_Contact(in1 := "2号梯当前楼层数", in2 := 9)
      wire#w10
      Contact( "2号梯9层上呼" )
   END_RUNG wire#w3
   RUNG wire#w10
      Contact( "2号梯9层内呼指示灯" )
   END_RUNG wire#w3
   RUNG wire#w1
      { S7_Templates := "SrcType := Int" } EQ_Contact(in1 := "2号梯当前楼层数", in2 := 10)
      Contact( "2号梯10层内呼指示灯" )
   END_RUNG wire#w3
   RUNG wire#w1
      I_Contact( "2号梯上行命令" )
   END_RUNG wire#w3
   // the same network as SCL:
   IF "2号梯上行接触器" AND "2号梯上平层信号" AND ((("2号梯当前楼层数" = 2) AND ("2号梯2层上呼" OR "2号梯2层内呼指示灯")) OR (("2号梯当前楼层数" = 3) AND ("2号梯3层上呼" OR "2号梯3层内呼指示灯")) OR (("2号梯当前楼层数" = 4) AND ("2号梯4层上呼" OR "2号梯4层内呼指示灯")) OR (("2号梯当前楼层数" = 5) AND ("2号梯5层上呼" OR "2号梯5层内呼指示灯")) OR (("2号梯当前楼层数" = 6) AND ("2号梯6层上呼" OR "2号梯6层内呼指示灯")) OR (("2号梯当前楼层数" = 7) AND ("2号梯7层上呼" OR "2号梯7层内呼指示灯")) OR (("2号梯当前楼层数" = 8) AND ("2号梯8层上呼" OR "2号梯8层内呼指示灯")) OR (("2号梯当前楼层数" = 9) AND ("2号梯9层上呼" OR "2号梯9层内呼指示灯")) OR (("2号梯当前楼层数" = 10) AND "2号梯10层内呼指示灯") OR NOT "2号梯上行命令") THEN
       "2号梯平层信号" := TRUE;
   END_IF;
END_REGION

REGION Network 2: 下行拦截电梯
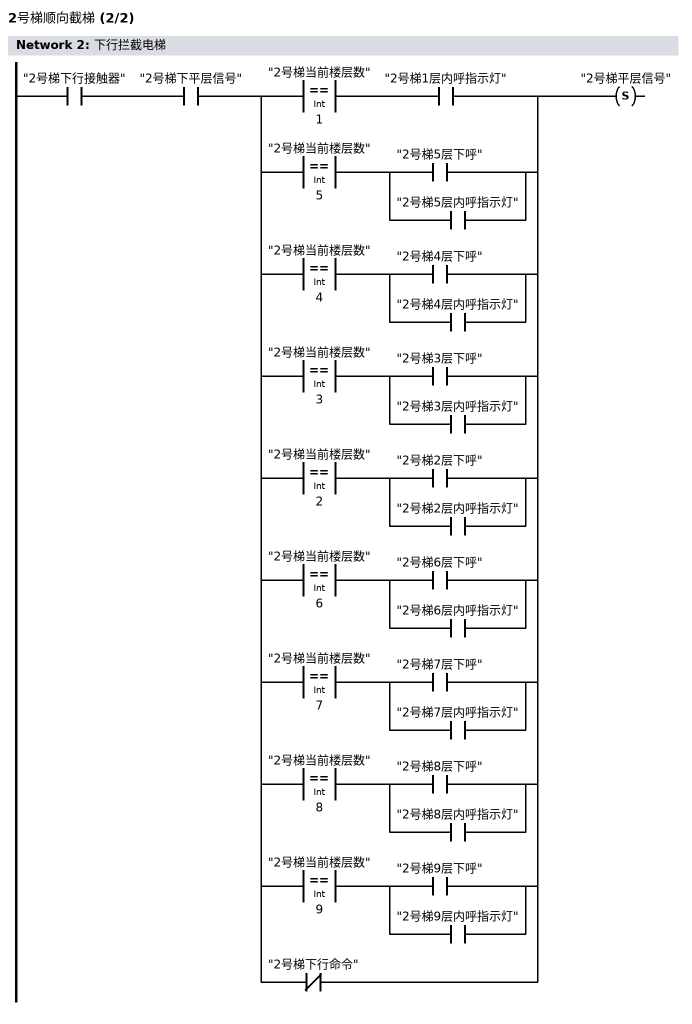
   RUNG wire#powerrail
      Contact( "2号梯下行接触器" )
      Contact( "2号梯下平层信号" )
      wire#w1
      { S7_Templates := "SrcType := Int" } EQ_Contact(in1 := "2号梯当前楼层数", in2 := 1)
      Contact( "2号梯1层内呼指示灯" )
      wire#w2
      S_Coil( "2号梯平层信号" )
   END_RUNG
   RUNG wire#w1
      { S7_Templates := "SrcType := Int" } EQ_Contact(in1 := "2号梯当前楼层数", in2 := 5)
      wire#w3
      Contact( "2号梯5层下呼" )
   END_RUNG wire#w2
   RUNG wire#w3
      Contact( "2号梯5层内呼指示灯" )
   END_RUNG wire#w2
   RUNG wire#w1
      { S7_Templates := "SrcType := Int" } EQ_Contact(in1 := "2号梯当前楼层数", in2 := 4)
      wire#w4
      Contact( "2号梯4层下呼" )
   END_RUNG wire#w2
   RUNG wire#w4
      Contact( "2号梯4层内呼指示灯" )
   END_RUNG wire#w2
   RUNG wire#w1
      { S7_Templates := "SrcType := Int" } EQ_Contact(in1 := "2号梯当前楼层数", in2 := 3)
      wire#w5
      Contact( "2号梯3层下呼" )
   END_RUNG wire#w2
   RUNG wire#w5
      Contact( "2号梯3层内呼指示灯" )
   END_RUNG wire#w2
   RUNG wire#w1
      { S7_Templates := "SrcType := Int" } EQ_Contact(in1 := "2号梯当前楼层数", in2 := 2)
      wire#w6
      Contact( "2号梯2层下呼" )
   END_RUNG wire#w2
   RUNG wire#w6
      Contact( "2号梯2层内呼指示灯" )
   END_RUNG wire#w2
   RUNG wire#w1
      { S7_Templates := "SrcType := Int" } EQ_Contact(in1 := "2号梯当前楼层数", in2 := 6)
      wire#w7
      Contact( "2号梯6层下呼" )
   END_RUNG wire#w2
   RUNG wire#w7
      Contact( "2号梯6层内呼指示灯" )
   END_RUNG wire#w2
   RUNG wire#w1
      { S7_Templates := "SrcType := Int" } EQ_Contact(in1 := "2号梯当前楼层数", in2 := 7)
      wire#w8
      Contact( "2号梯7层下呼" )
   END_RUNG wire#w2
   RUNG wire#w8
      Contact( "2号梯7层内呼指示灯" )
   END_RUNG wire#w2
   RUNG wire#w1
      { S7_Templates := "SrcType := Int" } EQ_Contact(in1 := "2号梯当前楼层数", in2 := 8)
      wire#w9
      Contact( "2号梯8层下呼" )
   END_RUNG wire#w2
   RUNG wire#w9
      Contact( "2号梯8层内呼指示灯" )
   END_RUNG wire#w2
   RUNG wire#w1
      { S7_Templates := "SrcType := Int" } EQ_Contact(in1 := "2号梯当前楼层数", in2 := 9)
      wire#w10
      Contact( "2号梯9层下呼" )
   END_RUNG wire#w2
   RUNG wire#w10
      Contact( "2号梯9层内呼指示灯" )
   END_RUNG wire#w2
   RUNG wire#w1
      I_Contact( "2号梯下行命令" )
   END_RUNG wire#w2
   // the same network as SCL:
   IF "2号梯下行接触器" AND "2号梯下平层信号" AND ((("2号梯当前楼层数" = 1) AND "2号梯1层内呼指示灯") OR (("2号梯当前楼层数" = 5) AND ("2号梯5层下呼" OR "2号梯5层内呼指示灯")) OR (("2号梯当前楼层数" = 4) AND ("2号梯4层下呼" OR "2号梯4层内呼指示灯")) OR (("2号梯当前楼层数" = 3) AND ("2号梯3层下呼" OR "2号梯3层内呼指示灯")) OR (("2号梯当前楼层数" = 2) AND ("2号梯2层下呼" OR "2号梯2层内呼指示灯")) OR (("2号梯当前楼层数" = 6) AND ("2号梯6层下呼" OR "2号梯6层内呼指示灯")) OR (("2号梯当前楼层数" = 7) AND ("2号梯7层下呼" OR "2号梯7层内呼指示灯")) OR (("2号梯当前楼层数" = 8) AND ("2号梯8层下呼" OR "2号梯8层内呼指示灯")) OR (("2号梯当前楼层数" = 9) AND ("2号梯9层下呼" OR "2号梯9层内呼指示灯")) OR NOT "2号梯下行命令") THEN
       "2号梯平层信号" := TRUE;
   END_IF;
END_REGION
END_FUNCTION

FUNCTION "3号梯顺向截梯" : Void   // FC38, LAD
{ S7_Optimized_Access := 'TRUE' }
VERSION : 0.1
BEGIN

REGION Network 1: 上行拦截电梯
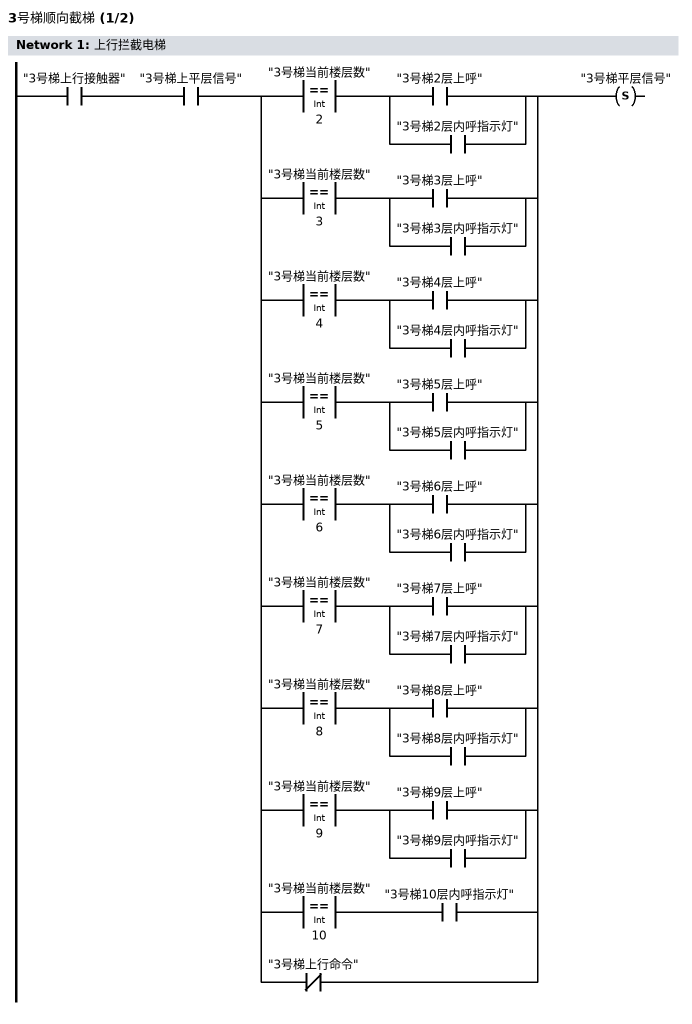
   RUNG wire#powerrail
      Contact( "3号梯上行接触器" )
      Contact( "3号梯上平层信号" )
      wire#w1
      { S7_Templates := "SrcType := Int" } EQ_Contact(in1 := "3号梯当前楼层数", in2 := 2)
      wire#w2
      Contact( "3号梯2层上呼" )
      wire#w3
      S_Coil( "3号梯平层信号" )
   END_RUNG
   RUNG wire#w2
      Contact( "3号梯2层内呼指示灯" )
   END_RUNG wire#w3
   RUNG wire#w1
      { S7_Templates := "SrcType := Int" } EQ_Contact(in1 := "3号梯当前楼层数", in2 := 3)
      wire#w4
      Contact( "3号梯3层上呼" )
   END_RUNG wire#w3
   RUNG wire#w4
      Contact( "3号梯3层内呼指示灯" )
   END_RUNG wire#w3
   RUNG wire#w1
      { S7_Templates := "SrcType := Int" } EQ_Contact(in1 := "3号梯当前楼层数", in2 := 4)
      wire#w5
      Contact( "3号梯4层上呼" )
   END_RUNG wire#w3
   RUNG wire#w5
      Contact( "3号梯4层内呼指示灯" )
   END_RUNG wire#w3
   RUNG wire#w1
      { S7_Templates := "SrcType := Int" } EQ_Contact(in1 := "3号梯当前楼层数", in2 := 5)
      wire#w6
      Contact( "3号梯5层上呼" )
   END_RUNG wire#w3
   RUNG wire#w6
      Contact( "3号梯5层内呼指示灯" )
   END_RUNG wire#w3
   RUNG wire#w1
      { S7_Templates := "SrcType := Int" } EQ_Contact(in1 := "3号梯当前楼层数", in2 := 6)
      wire#w7
      Contact( "3号梯6层上呼" )
   END_RUNG wire#w3
   RUNG wire#w7
      Contact( "3号梯6层内呼指示灯" )
   END_RUNG wire#w3
   RUNG wire#w1
      { S7_Templates := "SrcType := Int" } EQ_Contact(in1 := "3号梯当前楼层数", in2 := 7)
      wire#w8
      Contact( "3号梯7层上呼" )
   END_RUNG wire#w3
   RUNG wire#w8
      Contact( "3号梯7层内呼指示灯" )
   END_RUNG wire#w3
   RUNG wire#w1
      { S7_Templates := "SrcType := Int" } EQ_Contact(in1 := "3号梯当前楼层数", in2 := 8)
      wire#w9
      Contact( "3号梯8层上呼" )
   END_RUNG wire#w3
   RUNG wire#w9
      Contact( "3号梯8层内呼指示灯" )
   END_RUNG wire#w3
   RUNG wire#w1
      { S7_Templates := "SrcType := Int" } EQ_Contact(in1 := "3号梯当前楼层数", in2 := 9)
      wire#w10
      Contact( "3号梯9层上呼" )
   END_RUNG wire#w3
   RUNG wire#w10
      Contact( "3号梯9层内呼指示灯" )
   END_RUNG wire#w3
   RUNG wire#w1
      { S7_Templates := "SrcType := Int" } EQ_Contact(in1 := "3号梯当前楼层数", in2 := 10)
      Contact( "3号梯10层内呼指示灯" )
   END_RUNG wire#w3
   RUNG wire#w1
      I_Contact( "3号梯上行命令" )
   END_RUNG wire#w3
   // the same network as SCL:
   IF "3号梯上行接触器" AND "3号梯上平层信号" AND ((("3号梯当前楼层数" = 2) AND ("3号梯2层上呼" OR "3号梯2层内呼指示灯")) OR (("3号梯当前楼层数" = 3) AND ("3号梯3层上呼" OR "3号梯3层内呼指示灯")) OR (("3号梯当前楼层数" = 4) AND ("3号梯4层上呼" OR "3号梯4层内呼指示灯")) OR (("3号梯当前楼层数" = 5) AND ("3号梯5层上呼" OR "3号梯5层内呼指示灯")) OR (("3号梯当前楼层数" = 6) AND ("3号梯6层上呼" OR "3号梯6层内呼指示灯")) OR (("3号梯当前楼层数" = 7) AND ("3号梯7层上呼" OR "3号梯7层内呼指示灯")) OR (("3号梯当前楼层数" = 8) AND ("3号梯8层上呼" OR "3号梯8层内呼指示灯")) OR (("3号梯当前楼层数" = 9) AND ("3号梯9层上呼" OR "3号梯9层内呼指示灯")) OR (("3号梯当前楼层数" = 10) AND "3号梯10层内呼指示灯") OR NOT "3号梯上行命令") THEN
       "3号梯平层信号" := TRUE;
   END_IF;
END_REGION

REGION Network 2: 下行拦截电梯
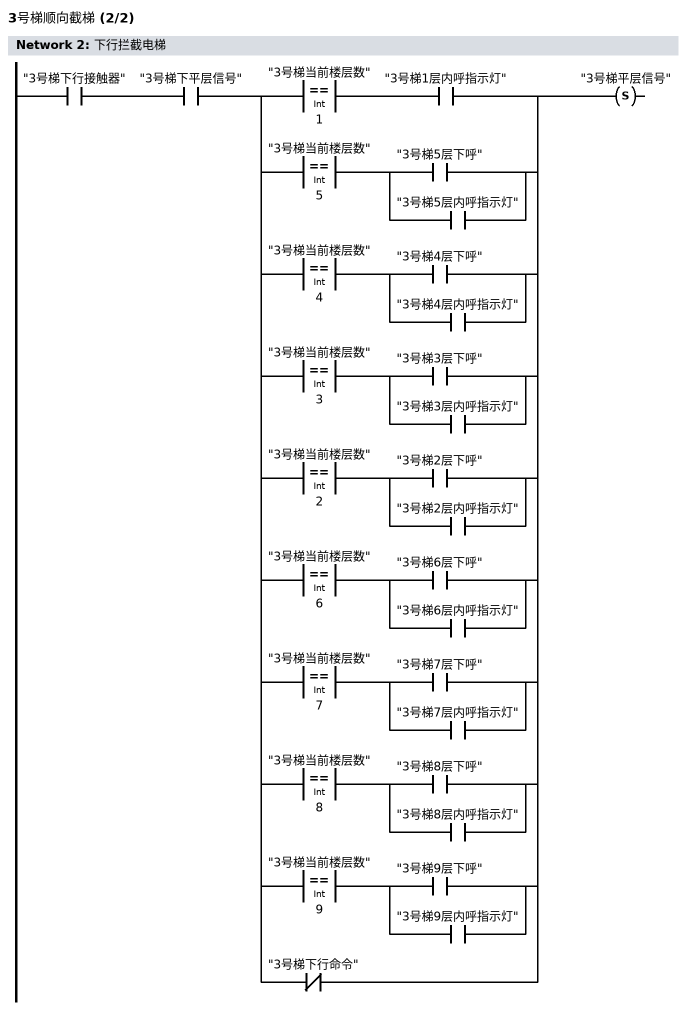
   RUNG wire#powerrail
      Contact( "3号梯下行接触器" )
      Contact( "3号梯下平层信号" )
      wire#w1
      { S7_Templates := "SrcType := Int" } EQ_Contact(in1 := "3号梯当前楼层数", in2 := 1)
      Contact( "3号梯1层内呼指示灯" )
      wire#w2
      S_Coil( "3号梯平层信号" )
   END_RUNG
   RUNG wire#w1
      { S7_Templates := "SrcType := Int" } EQ_Contact(in1 := "3号梯当前楼层数", in2 := 5)
      wire#w3
      Contact( "3号梯5层下呼" )
   END_RUNG wire#w2
   RUNG wire#w3
      Contact( "3号梯5层内呼指示灯" )
   END_RUNG wire#w2
   RUNG wire#w1
      { S7_Templates := "SrcType := Int" } EQ_Contact(in1 := "3号梯当前楼层数", in2 := 4)
      wire#w4
      Contact( "3号梯4层下呼" )
   END_RUNG wire#w2
   RUNG wire#w4
      Contact( "3号梯4层内呼指示灯" )
   END_RUNG wire#w2
   RUNG wire#w1
      { S7_Templates := "SrcType := Int" } EQ_Contact(in1 := "3号梯当前楼层数", in2 := 3)
      wire#w5
      Contact( "3号梯3层下呼" )
   END_RUNG wire#w2
   RUNG wire#w5
      Contact( "3号梯3层内呼指示灯" )
   END_RUNG wire#w2
   RUNG wire#w1
      { S7_Templates := "SrcType := Int" } EQ_Contact(in1 := "3号梯当前楼层数", in2 := 2)
      wire#w6
      Contact( "3号梯2层下呼" )
   END_RUNG wire#w2
   RUNG wire#w6
      Contact( "3号梯2层内呼指示灯" )
   END_RUNG wire#w2
   RUNG wire#w1
      { S7_Templates := "SrcType := Int" } EQ_Contact(in1 := "3号梯当前楼层数", in2 := 6)
      wire#w7
      Contact( "3号梯6层下呼" )
   END_RUNG wire#w2
   RUNG wire#w7
      Contact( "3号梯6层内呼指示灯" )
   END_RUNG wire#w2
   RUNG wire#w1
      { S7_Templates := "SrcType := Int" } EQ_Contact(in1 := "3号梯当前楼层数", in2 := 7)
      wire#w8
      Contact( "3号梯7层下呼" )
   END_RUNG wire#w2
   RUNG wire#w8
      Contact( "3号梯7层内呼指示灯" )
   END_RUNG wire#w2
   RUNG wire#w1
      { S7_Templates := "SrcType := Int" } EQ_Contact(in1 := "3号梯当前楼层数", in2 := 8)
      wire#w9
      Contact( "3号梯8层下呼" )
   END_RUNG wire#w2
   RUNG wire#w9
      Contact( "3号梯8层内呼指示灯" )
   END_RUNG wire#w2
   RUNG wire#w1
      { S7_Templates := "SrcType := Int" } EQ_Contact(in1 := "3号梯当前楼层数", in2 := 9)
      wire#w10
      Contact( "3号梯9层下呼" )
   END_RUNG wire#w2
   RUNG wire#w10
      Contact( "3号梯9层内呼指示灯" )
   END_RUNG wire#w2
   RUNG wire#w1
      I_Contact( "3号梯下行命令" )
   END_RUNG wire#w2
   // the same network as SCL:
   IF "3号梯下行接触器" AND "3号梯下平层信号" AND ((("3号梯当前楼层数" = 1) AND "3号梯1层内呼指示灯") OR (("3号梯当前楼层数" = 5) AND ("3号梯5层下呼" OR "3号梯5层内呼指示灯")) OR (("3号梯当前楼层数" = 4) AND ("3号梯4层下呼" OR "3号梯4层内呼指示灯")) OR (("3号梯当前楼层数" = 3) AND ("3号梯3层下呼" OR "3号梯3层内呼指示灯")) OR (("3号梯当前楼层数" = 2) AND ("3号梯2层下呼" OR "3号梯2层内呼指示灯")) OR (("3号梯当前楼层数" = 6) AND ("3号梯6层下呼" OR "3号梯6层内呼指示灯")) OR (("3号梯当前楼层数" = 7) AND ("3号梯7层下呼" OR "3号梯7层内呼指示灯")) OR (("3号梯当前楼层数" = 8) AND ("3号梯8层下呼" OR "3号梯8层内呼指示灯")) OR (("3号梯当前楼层数" = 9) AND ("3号梯9层下呼" OR "3号梯9层内呼指示灯")) OR NOT "3号梯下行命令") THEN
       "3号梯平层信号" := TRUE;
   END_IF;
END_REGION
END_FUNCTION

FUNCTION "2号梯轿内指示灯控制" : Void   // FC39, LAD
{ S7_Optimized_Access := 'TRUE' }
VERSION : 0.1
   VAR_TEMP   // added for the SCL form of the ladder/FBD networks
      _w1 : Bool;
      _w2 : Bool;
   END_VAR
BEGIN

REGION Network 1: 平层灭灯
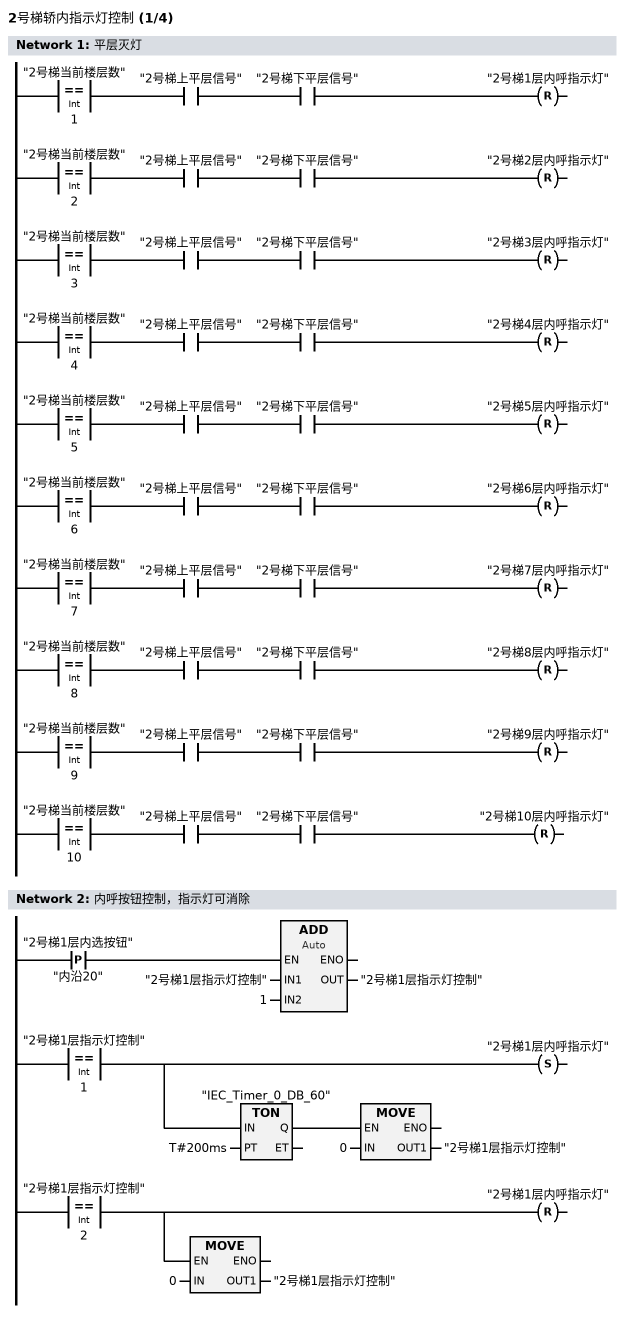
   RUNG wire#powerrail
      { S7_Templates := "SrcType := Int" } EQ_Contact(in1 := "2号梯当前楼层数", in2 := 1)
      Contact( "2号梯上平层信号" )
      Contact( "2号梯下平层信号" )
      R_Coil( "2号梯1层内呼指示灯" )
   END_RUNG
   RUNG wire#powerrail
      { S7_Templates := "SrcType := Int" } EQ_Contact(in1 := "2号梯当前楼层数", in2 := 2)
      Contact( "2号梯上平层信号" )
      Contact( "2号梯下平层信号" )
      R_Coil( "2号梯2层内呼指示灯" )
   END_RUNG
   RUNG wire#powerrail
      { S7_Templates := "SrcType := Int" } EQ_Contact(in1 := "2号梯当前楼层数", in2 := 3)
      Contact( "2号梯上平层信号" )
      Contact( "2号梯下平层信号" )
      R_Coil( "2号梯3层内呼指示灯" )
   END_RUNG
   RUNG wire#powerrail
      { S7_Templates := "SrcType := Int" } EQ_Contact(in1 := "2号梯当前楼层数", in2 := 4)
      Contact( "2号梯上平层信号" )
      Contact( "2号梯下平层信号" )
      R_Coil( "2号梯4层内呼指示灯" )
   END_RUNG
   RUNG wire#powerrail
      { S7_Templates := "SrcType := Int" } EQ_Contact(in1 := "2号梯当前楼层数", in2 := 5)
      Contact( "2号梯上平层信号" )
      Contact( "2号梯下平层信号" )
      R_Coil( "2号梯5层内呼指示灯" )
   END_RUNG
   RUNG wire#powerrail
      { S7_Templates := "SrcType := Int" } EQ_Contact(in1 := "2号梯当前楼层数", in2 := 6)
      Contact( "2号梯上平层信号" )
      Contact( "2号梯下平层信号" )
      R_Coil( "2号梯6层内呼指示灯" )
   END_RUNG
   RUNG wire#powerrail
      { S7_Templates := "SrcType := Int" } EQ_Contact(in1 := "2号梯当前楼层数", in2 := 7)
      Contact( "2号梯上平层信号" )
      Contact( "2号梯下平层信号" )
      R_Coil( "2号梯7层内呼指示灯" )
   END_RUNG
   RUNG wire#powerrail
      { S7_Templates := "SrcType := Int" } EQ_Contact(in1 := "2号梯当前楼层数", in2 := 8)
      Contact( "2号梯上平层信号" )
      Contact( "2号梯下平层信号" )
      R_Coil( "2号梯8层内呼指示灯" )
   END_RUNG
   RUNG wire#powerrail
      { S7_Templates := "SrcType := Int" } EQ_Contact(in1 := "2号梯当前楼层数", in2 := 9)
      Contact( "2号梯上平层信号" )
      Contact( "2号梯下平层信号" )
      R_Coil( "2号梯9层内呼指示灯" )
   END_RUNG
   RUNG wire#powerrail
      { S7_Templates := "SrcType := Int" } EQ_Contact(in1 := "2号梯当前楼层数", in2 := 10)
      Contact( "2号梯上平层信号" )
      Contact( "2号梯下平层信号" )
      R_Coil( "2号梯10层内呼指示灯" )
   END_RUNG
   // the same network as SCL:
   IF ("2号梯当前楼层数" = 1) AND "2号梯上平层信号" AND "2号梯下平层信号" THEN "2号梯1层内呼指示灯" := FALSE; END_IF;
   IF ("2号梯当前楼层数" = 2) AND "2号梯上平层信号" AND "2号梯下平层信号" THEN "2号梯2层内呼指示灯" := FALSE; END_IF;
   IF ("2号梯当前楼层数" = 3) AND "2号梯上平层信号" AND "2号梯下平层信号" THEN "2号梯3层内呼指示灯" := FALSE; END_IF;
   IF ("2号梯当前楼层数" = 4) AND "2号梯上平层信号" AND "2号梯下平层信号" THEN "2号梯4层内呼指示灯" := FALSE; END_IF;
   IF ("2号梯当前楼层数" = 5) AND "2号梯上平层信号" AND "2号梯下平层信号" THEN "2号梯5层内呼指示灯" := FALSE; END_IF;
   IF ("2号梯当前楼层数" = 6) AND "2号梯上平层信号" AND "2号梯下平层信号" THEN "2号梯6层内呼指示灯" := FALSE; END_IF;
   IF ("2号梯当前楼层数" = 7) AND "2号梯上平层信号" AND "2号梯下平层信号" THEN "2号梯7层内呼指示灯" := FALSE; END_IF;
   IF ("2号梯当前楼层数" = 8) AND "2号梯上平层信号" AND "2号梯下平层信号" THEN "2号梯8层内呼指示灯" := FALSE; END_IF;
   IF ("2号梯当前楼层数" = 9) AND "2号梯上平层信号" AND "2号梯下平层信号" THEN "2号梯9层内呼指示灯" := FALSE; END_IF;
   IF ("2号梯当前楼层数" = 10) AND "2号梯上平层信号" AND "2号梯下平层信号" THEN "2号梯10层内呼指示灯" := FALSE; END_IF;
END_REGION

REGION Network 2: 内呼按钮控制，指示灯可消除
   #_w1 := "2号梯1层内选按钮" AND NOT "内沿20";   // rising edge of "2号梯1层内选按钮"
   "内沿20" := "2号梯1层内选按钮";
   IF #_w1 THEN "2号梯1层指示灯控制" := "2号梯1层指示灯控制" + 1; END_IF;
   #_w2 := "2号梯1层指示灯控制" = 1;
   IF #_w2 THEN "2号梯1层内呼指示灯" := TRUE; END_IF;
   "IEC_Timer_0_DB_60".TON(IN := #_w2, PT := T#200ms);
   IF "IEC_Timer_0_DB_60".Q THEN "2号梯1层指示灯控制" := 0; END_IF;
   IF "2号梯1层指示灯控制" = 2 THEN
       "2号梯1层内呼指示灯" := FALSE;
       "2号梯1层指示灯控制" := 0;
   END_IF;
END_REGION

REGION Network 3: 内呼按钮控制，指示灯可消除
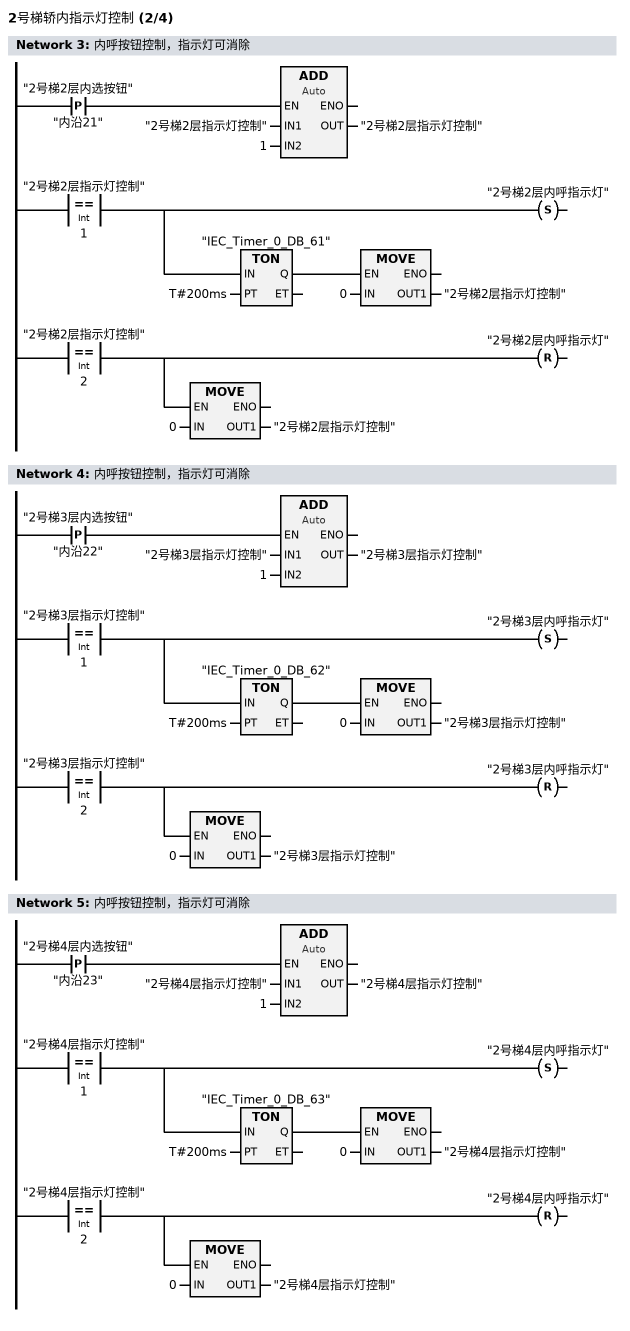
   #_w1 := "2号梯2层内选按钮" AND NOT "内沿21";   // rising edge of "2号梯2层内选按钮"
   "内沿21" := "2号梯2层内选按钮";
   IF #_w1 THEN "2号梯2层指示灯控制" := "2号梯2层指示灯控制" + 1; END_IF;
   #_w2 := "2号梯2层指示灯控制" = 1;
   IF #_w2 THEN "2号梯2层内呼指示灯" := TRUE; END_IF;
   "IEC_Timer_0_DB_61".TON(IN := #_w2, PT := T#200ms);
   IF "IEC_Timer_0_DB_61".Q THEN "2号梯2层指示灯控制" := 0; END_IF;
   IF "2号梯2层指示灯控制" = 2 THEN
       "2号梯2层内呼指示灯" := FALSE;
       "2号梯2层指示灯控制" := 0;
   END_IF;
END_REGION

REGION Network 4: 内呼按钮控制，指示灯可消除
   #_w1 := "2号梯3层内选按钮" AND NOT "内沿22";   // rising edge of "2号梯3层内选按钮"
   "内沿22" := "2号梯3层内选按钮";
   IF #_w1 THEN "2号梯3层指示灯控制" := "2号梯3层指示灯控制" + 1; END_IF;
   #_w2 := "2号梯3层指示灯控制" = 1;
   IF #_w2 THEN "2号梯3层内呼指示灯" := TRUE; END_IF;
   "IEC_Timer_0_DB_62".TON(IN := #_w2, PT := T#200ms);
   IF "IEC_Timer_0_DB_62".Q THEN "2号梯3层指示灯控制" := 0; END_IF;
   IF "2号梯3层指示灯控制" = 2 THEN
       "2号梯3层内呼指示灯" := FALSE;
       "2号梯3层指示灯控制" := 0;
   END_IF;
END_REGION

REGION Network 5: 内呼按钮控制，指示灯可消除
   #_w1 := "2号梯4层内选按钮" AND NOT "内沿23";   // rising edge of "2号梯4层内选按钮"
   "内沿23" := "2号梯4层内选按钮";
   IF #_w1 THEN "2号梯4层指示灯控制" := "2号梯4层指示灯控制" + 1; END_IF;
   #_w2 := "2号梯4层指示灯控制" = 1;
   IF #_w2 THEN "2号梯4层内呼指示灯" := TRUE; END_IF;
   "IEC_Timer_0_DB_63".TON(IN := #_w2, PT := T#200ms);
   IF "IEC_Timer_0_DB_63".Q THEN "2号梯4层指示灯控制" := 0; END_IF;
   IF "2号梯4层指示灯控制" = 2 THEN
       "2号梯4层内呼指示灯" := FALSE;
       "2号梯4层指示灯控制" := 0;
   END_IF;
END_REGION

REGION Network 6: 内呼按钮控制，指示灯可消除
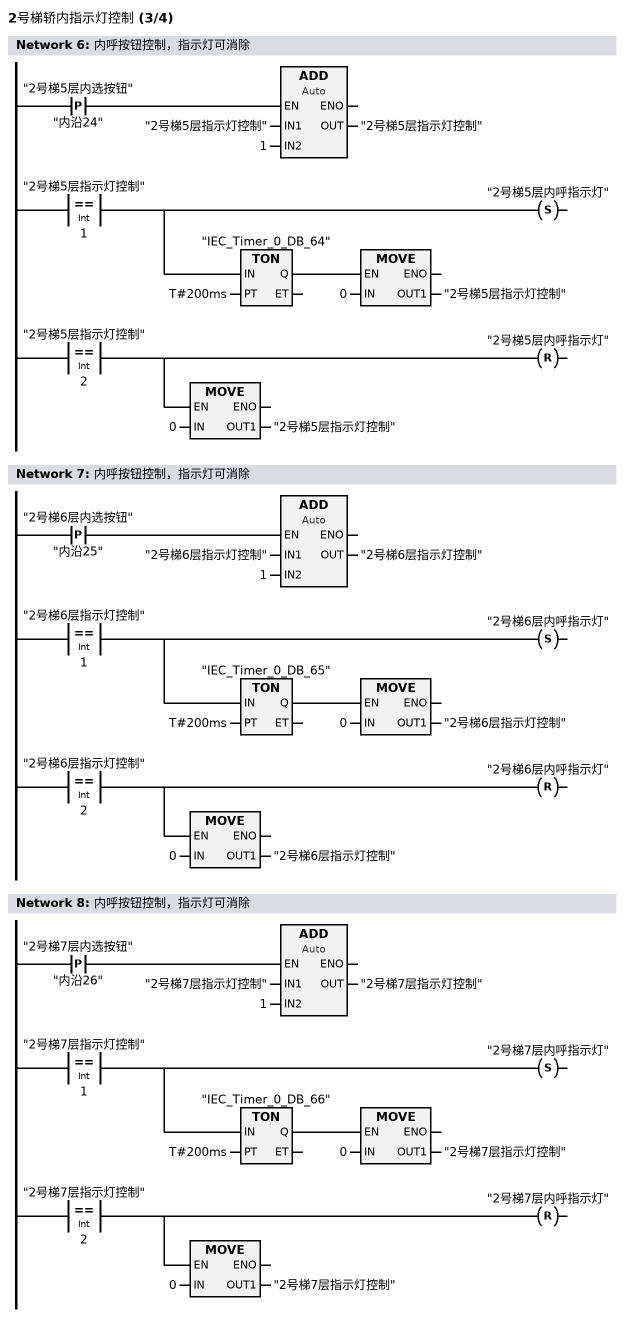
   #_w1 := "2号梯5层内选按钮" AND NOT "内沿24";   // rising edge of "2号梯5层内选按钮"
   "内沿24" := "2号梯5层内选按钮";
   IF #_w1 THEN "2号梯5层指示灯控制" := "2号梯5层指示灯控制" + 1; END_IF;
   #_w2 := "2号梯5层指示灯控制" = 1;
   IF #_w2 THEN "2号梯5层内呼指示灯" := TRUE; END_IF;
   "IEC_Timer_0_DB_64".TON(IN := #_w2, PT := T#200ms);
   IF "IEC_Timer_0_DB_64".Q THEN "2号梯5层指示灯控制" := 0; END_IF;
   IF "2号梯5层指示灯控制" = 2 THEN
       "2号梯5层内呼指示灯" := FALSE;
       "2号梯5层指示灯控制" := 0;
   END_IF;
END_REGION

REGION Network 7: 内呼按钮控制，指示灯可消除
   #_w1 := "2号梯6层内选按钮" AND NOT "内沿25";   // rising edge of "2号梯6层内选按钮"
   "内沿25" := "2号梯6层内选按钮";
   IF #_w1 THEN "2号梯6层指示灯控制" := "2号梯6层指示灯控制" + 1; END_IF;
   #_w2 := "2号梯6层指示灯控制" = 1;
   IF #_w2 THEN "2号梯6层内呼指示灯" := TRUE; END_IF;
   "IEC_Timer_0_DB_65".TON(IN := #_w2, PT := T#200ms);
   IF "IEC_Timer_0_DB_65".Q THEN "2号梯6层指示灯控制" := 0; END_IF;
   IF "2号梯6层指示灯控制" = 2 THEN
       "2号梯6层内呼指示灯" := FALSE;
       "2号梯6层指示灯控制" := 0;
   END_IF;
END_REGION

REGION Network 8: 内呼按钮控制，指示灯可消除
   #_w1 := "2号梯7层内选按钮" AND NOT "内沿26";   // rising edge of "2号梯7层内选按钮"
   "内沿26" := "2号梯7层内选按钮";
   IF #_w1 THEN "2号梯7层指示灯控制" := "2号梯7层指示灯控制" + 1; END_IF;
   #_w2 := "2号梯7层指示灯控制" = 1;
   IF #_w2 THEN "2号梯7层内呼指示灯" := TRUE; END_IF;
   "IEC_Timer_0_DB_66".TON(IN := #_w2, PT := T#200ms);
   IF "IEC_Timer_0_DB_66".Q THEN "2号梯7层指示灯控制" := 0; END_IF;
   IF "2号梯7层指示灯控制" = 2 THEN
       "2号梯7层内呼指示灯" := FALSE;
       "2号梯7层指示灯控制" := 0;
   END_IF;
END_REGION

REGION Network 9: 内呼按钮控制，指示灯可消除
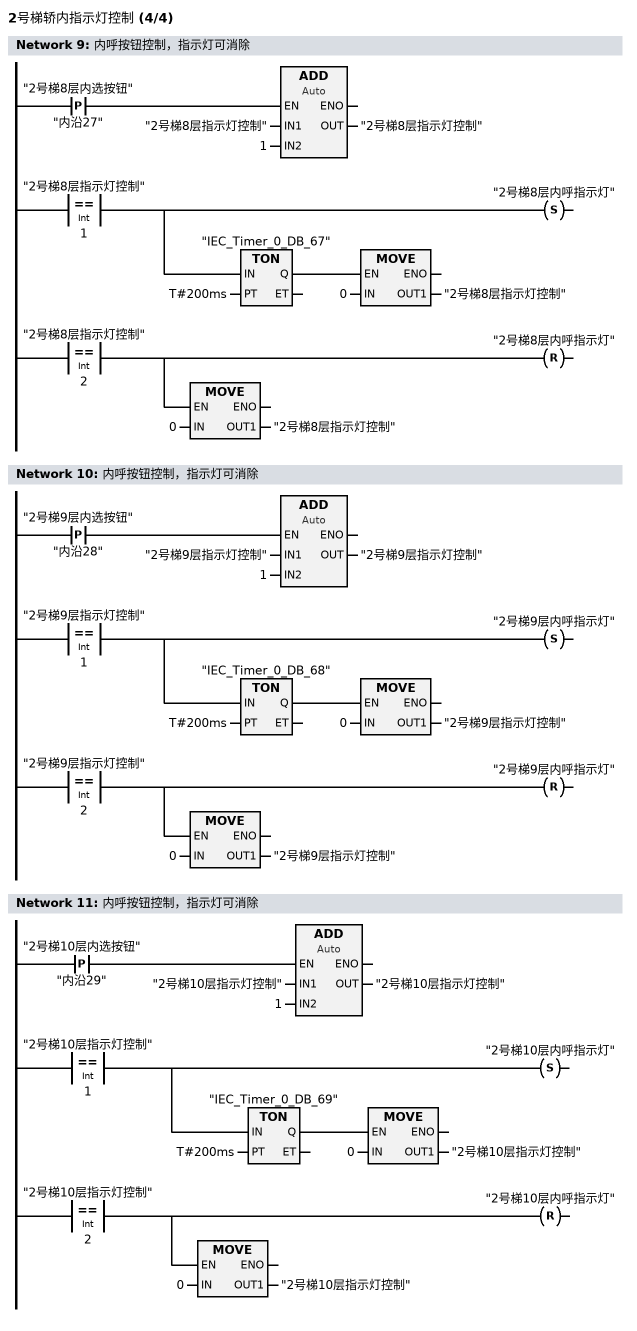
   #_w1 := "2号梯8层内选按钮" AND NOT "内沿27";   // rising edge of "2号梯8层内选按钮"
   "内沿27" := "2号梯8层内选按钮";
   IF #_w1 THEN "2号梯8层指示灯控制" := "2号梯8层指示灯控制" + 1; END_IF;
   #_w2 := "2号梯8层指示灯控制" = 1;
   IF #_w2 THEN "2号梯8层内呼指示灯" := TRUE; END_IF;
   "IEC_Timer_0_DB_67".TON(IN := #_w2, PT := T#200ms);
   IF "IEC_Timer_0_DB_67".Q THEN "2号梯8层指示灯控制" := 0; END_IF;
   IF "2号梯8层指示灯控制" = 2 THEN
       "2号梯8层内呼指示灯" := FALSE;
       "2号梯8层指示灯控制" := 0;
   END_IF;
END_REGION

REGION Network 10: 内呼按钮控制，指示灯可消除
   #_w1 := "2号梯9层内选按钮" AND NOT "内沿28";   // rising edge of "2号梯9层内选按钮"
   "内沿28" := "2号梯9层内选按钮";
   IF #_w1 THEN "2号梯9层指示灯控制" := "2号梯9层指示灯控制" + 1; END_IF;
   #_w2 := "2号梯9层指示灯控制" = 1;
   IF #_w2 THEN "2号梯9层内呼指示灯" := TRUE; END_IF;
   "IEC_Timer_0_DB_68".TON(IN := #_w2, PT := T#200ms);
   IF "IEC_Timer_0_DB_68".Q THEN "2号梯9层指示灯控制" := 0; END_IF;
   IF "2号梯9层指示灯控制" = 2 THEN
       "2号梯9层内呼指示灯" := FALSE;
       "2号梯9层指示灯控制" := 0;
   END_IF;
END_REGION

REGION Network 11: 内呼按钮控制，指示灯可消除
   #_w1 := "2号梯10层内选按钮" AND NOT "内沿29";   // rising edge of "2号梯10层内选按钮"
   "内沿29" := "2号梯10层内选按钮";
   IF #_w1 THEN "2号梯10层指示灯控制" := "2号梯10层指示灯控制" + 1; END_IF;
   #_w2 := "2号梯10层指示灯控制" = 1;
   IF #_w2 THEN "2号梯10层内呼指示灯" := TRUE; END_IF;
   "IEC_Timer_0_DB_69".TON(IN := #_w2, PT := T#200ms);
   IF "IEC_Timer_0_DB_69".Q THEN "2号梯10层指示灯控制" := 0; END_IF;
   IF "2号梯10层指示灯控制" = 2 THEN
       "2号梯10层内呼指示灯" := FALSE;
       "2号梯10层指示灯控制" := 0;
   END_IF;
END_REGION
END_FUNCTION

FUNCTION "3号梯轿内指示灯控制" : Void   // FC40, LAD
{ S7_Optimized_Access := 'TRUE' }
VERSION : 0.1
   VAR_TEMP   // added for the SCL form of the ladder/FBD networks
      _w1 : Bool;
      _w2 : Bool;
   END_VAR
BEGIN

REGION Network 1: 平层灭灯
